  MoveL 2659 to (228.12, 35.85, 50.44) mm, rotated rx -180 ry 0 rz -180 deg; joints [-156.181, -75.797, -46.821, 39.316, 39.597, -32.253]
  MoveL 2660 to (228.12, 35.85, 50.44) mm, rotated rx -180 ry 0 rz -180 deg; joints [-156.181, -75.797, -46.821, 39.316, 39.597, -32.253]
  Call Extruder(588.66808)
  MoveL 2661 to (228.37, 35.9, 50.44) mm, rotated rx 180 ry 0 rz -180 deg; joints [-156.187, -75.828, -46.752, 39.337, 39.565, -32.285]
  MoveL 2662 to (228.37, 35.9, 50.44) mm, rotated rx 180 ry 0 rz -180 deg; joints [-156.187, -75.828, -46.752, 39.337, 39.565, -32.285]
  Call Extruder(588.80265)
  MoveL 2663 to (228.61, 35.95, 50.44) mm, rotated rx -180 ry 0 rz 180 deg; joints [-156.192, -75.86, -46.683, 39.359, 39.533, -32.317]
  MoveL 2664 to (228.61, 35.95, 50.44) mm, rotated rx -180 ry 0 rz 180 deg; joints [-156.192, -75.86, -46.683, 39.359, 39.533, -32.317]
  Call Extruder(588.88871)
  MoveL 2665 to (228.77, 35.98, 50.44) mm, rotated rx -180 ry 0 rz 180 deg; joints [-156.196, -75.88, -46.639, 39.373, 39.513, -32.338]
  MoveL 2666 to (228.77, 35.98, 50.44) mm, rotated rx -180 ry 0 rz 180 deg; joints [-156.196, -75.88, -46.639, 39.373, 39.513, -32.338]
  Call Extruder(589.00224)
  MoveL 2667 to (228.97, 36.02, 50.44) mm, rotated rx 180 ry 0 rz -180 deg; joints [-156.2, -75.906, -46.581, 39.391, 39.486, -32.365]
  MoveL 2668 to (228.97, 36.02, 50.44) mm, rotated rx 180 ry 0 rz -180 deg; joints [-156.2, -75.906, -46.581, 39.391, 39.486, -32.365]
  Call Extruder(589.11625)
  MoveL 2669 to (229.18, 36.06, 50.44) mm, rotated rx 180 ry 0 rz 180 deg; joints [-156.205, -75.932, -46.523, 39.41, 39.458, -32.392]
  MoveL 2670 to (229.18, 36.06, 50.44) mm, rotated rx 180 ry 0 rz 180 deg; joints [-156.205, -75.932, -46.523, 39.41, 39.458, -32.392]
  Call Extruder(589.23074)
  MoveL 2671 to (229.38, 36.1, 50.44) mm, rotated rx 180 ry 0 rz 180 deg; joints [-156.21, -75.958, -46.465, 39.428, 39.431, -32.419]
  MoveL 2672 to (229.38, 36.1, 50.44) mm, rotated rx 180 ry 0 rz 180 deg; joints [-156.21, -75.958, -46.465, 39.428, 39.431, -32.419]
  Call Extruder(589.35620)
  MoveL 2673 to (229.6, 36.16, 50.44) mm, rotated rx 180 ry 0 rz 180 deg; joints [-156.213, -75.988, -46.4, 39.451, 39.403, -32.451]
  MoveL 2674 to (229.6, 36.16, 50.44) mm, rotated rx 180 ry 0 rz 180 deg; joints [-156.213, -75.988, -46.4, 39.451, 39.403, -32.451]
  Call Extruder(589.48218)
  MoveL 2675 to (229.82, 36.23, 50.44) mm, rotated rx 180 ry 0 rz 180 deg; joints [-156.215, -76.017, -46.335, 39.475, 39.374, -32.483]
  MoveL 2676 to (229.82, 36.23, 50.44) mm, rotated rx 180 ry 0 rz 180 deg; joints [-156.215, -76.017, -46.335, 39.475, 39.374, -32.483]
  Call Extruder(589.60868)
  MoveL 2677 to (230.04, 36.29, 50.44) mm, rotated rx 180 ry 0 rz 180 deg; joints [-156.218, -76.046, -46.271, 39.498, 39.345, -32.516]
  MoveL 2678 to (230.04, 36.29, 50.44) mm, rotated rx 180 ry 0 rz 180 deg; joints [-156.218, -76.046, -46.271, 39.498, 39.345, -32.516]
  Call Extruder(589.73571)
  MoveL 2679 to (230.26, 36.36, 50.44) mm, rotated rx -180 ry 0 rz 180 deg; joints [-156.221, -76.076, -46.206, 39.522, 39.316, -32.549]
  MoveL 2680 to (230.26, 36.36, 50.44) mm, rotated rx -180 ry 0 rz 180 deg; joints [-156.221, -76.076, -46.206, 39.522, 39.316, -32.549]
  Call Extruder(589.86325)
  MoveL 2681 to (230.48, 36.42, 50.44) mm, rotated rx 180 ry 0 rz -180 deg; joints [-156.224, -76.105, -46.141, 39.546, 39.287, -32.581]
  MoveL 2682 to (230.48, 36.42, 50.44) mm, rotated rx 180 ry 0 rz -180 deg; joints [-156.224, -76.105, -46.141, 39.546, 39.287, -32.581]
  Call Extruder(589.99132)
  MoveL 2683 to (230.69, 36.49, 50.44) mm, rotated rx 180 ry 0 rz -180 deg; joints [-156.227, -76.135, -46.076, 39.57, 39.258, -32.614]
  MoveL 2684 to (230.69, 36.49, 50.44) mm, rotated rx 180 ry 0 rz -180 deg; joints [-156.227, -76.135, -46.076, 39.57, 39.258, -32.614]
  Call Extruder(590.10322)
  MoveL 2685 to (230.88, 36.55, 50.44) mm, rotated rx -180 ry 0 rz 180 deg; joints [-156.229, -76.161, -46.019, 39.591, 39.233, -32.643]
  MoveL 2686 to (230.88, 36.55, 50.44) mm, rotated rx -180 ry 0 rz 180 deg; joints [-156.229, -76.161, -46.019, 39.591, 39.233, -32.643]
  Call Extruder(590.21556)
  MoveL 2687 to (231.07, 36.61, 50.44) mm, rotated rx 180 ry 0 rz 180 deg; joints [-156.231, -76.186, -45.962, 39.613, 39.208, -32.672]
  MoveL 2688 to (231.07, 36.61, 50.44) mm, rotated rx 180 ry 0 rz 180 deg; joints [-156.231, -76.186, -45.962, 39.613, 39.208, -32.672]
  Call Extruder(590.32835)
  MoveL 2689 to (231.26, 36.67, 50.44) mm, rotated rx 180 ry 0 rz -180 deg; joints [-156.233, -76.212, -45.905, 39.634, 39.183, -32.702]
  MoveL 2690 to (231.26, 36.67, 50.44) mm, rotated rx 180 ry 0 rz -180 deg; joints [-156.233, -76.212, -45.905, 39.634, 39.183, -32.702]
  Call Extruder(590.44158)
  MoveL 2691 to (231.45, 36.73, 50.44) mm, rotated rx -180 ry 0 rz 180 deg; joints [-156.235, -76.238, -45.848, 39.656, 39.158, -32.731]
  MoveL 2692 to (231.45, 36.73, 50.44) mm, rotated rx -180 ry 0 rz 180 deg; joints [-156.235, -76.238, -45.848, 39.656, 39.158, -32.731]
  Call Extruder(590.55526)
  MoveL 2693 to (231.64, 36.79, 50.44) mm, rotated rx 180 ry 0 rz 180 deg; joints [-156.237, -76.264, -45.792, 39.678, 39.133, -32.76]
  MoveL 2694 to (231.64, 36.79, 50.44) mm, rotated rx 180 ry 0 rz 180 deg; joints [-156.237, -76.264, -45.792, 39.678, 39.133, -32.76]
  Call Extruder(590.73722)
  MoveL 2695 to (231.93, 36.91, 50.44) mm, rotated rx 180 ry 0 rz 180 deg; joints [-156.238, -76.306, -45.7, 39.716, 39.095, -32.81]
  MoveL 2696 to (231.93, 36.91, 50.44) mm, rotated rx 180 ry 0 rz 180 deg; joints [-156.238, -76.306, -45.7, 39.716, 39.095, -32.81]
  Call Extruder(590.91994)
  MoveL 2697 to (232.22, 37.03, 50.44) mm, rotated rx 180 ry 0 rz 180 deg; joints [-156.238, -76.347, -45.609, 39.754, 39.056, -32.86]
  MoveL 2698 to (232.22, 37.03, 50.44) mm, rotated rx 180 ry 0 rz 180 deg; joints [-156.238, -76.347, -45.609, 39.754, 39.056, -32.86]
  Call Extruder(591.09035)
  MoveL 2699 to (232.49, 37.15, 50.44) mm, rotated rx 180 ry 0 rz 180 deg; joints [-156.239, -76.386, -45.524, 39.79, 39.02, -32.906]
  MoveL 2700 to (232.49, 37.15, 50.44) mm, rotated rx 180 ry 0 rz 180 deg; joints [-156.239, -76.386, -45.524, 39.79, 39.02, -32.906]
  Call Extruder(591.24835)
  MoveL 2701 to (232.74, 37.26, 50.44) mm, rotated rx 180 ry 0 rz 180 deg; joints [-156.239, -76.422, -45.445, 39.824, 38.987, -32.95]
  MoveL 2702 to (232.74, 37.26, 50.44) mm, rotated rx 180 ry 0 rz 180 deg; joints [-156.239, -76.422, -45.445, 39.824, 38.987, -32.95]
  Call Extruder(591.40695)
  MoveL 2703 to (232.99, 37.36, 50.44) mm, rotated rx -180 ry 0 rz -180 deg; joints [-156.239, -76.458, -45.366, 39.858, 38.954, -32.993]
  MoveL 2704 to (232.99, 37.36, 50.44) mm, rotated rx -180 ry 0 rz -180 deg; joints [-156.239, -76.458, -45.366, 39.858, 38.954, -32.993]
  Call Extruder(591.61312)
  MoveL 2705 to (233.29, 37.54, 50.44) mm, rotated rx 180 ry 0 rz 180 deg; joints [-156.236, -76.504, -45.264, 39.906, 38.913, -33.054]
  MoveL 2706 to (233.29, 37.54, 50.44) mm, rotated rx 180 ry 0 rz 180 deg; joints [-156.236, -76.504, -45.264, 39.906, 38.913, -33.054]
  Call Extruder(591.82006)
  MoveL 2707 to (233.6, 37.71, 50.44) mm, rotated rx 180 ry 0 rz 180 deg; joints [-156.232, -76.55, -45.162, 39.956, 38.873, -33.114]
  MoveL 2708 to (233.6, 37.71, 50.44) mm, rotated rx 180 ry 0 rz 180 deg; joints [-156.232, -76.55, -45.162, 39.956, 38.873, -33.114]
  Call Extruder(592.02779)
  MoveL 2709 to (233.9, 37.89, 50.44) mm, rotated rx 180 ry 0 rz 180 deg; joints [-156.228, -76.597, -45.061, 40.005, 38.832, -33.175]
  MoveL 2710 to (233.9, 37.89, 50.44) mm, rotated rx 180 ry 0 rz 180 deg; joints [-156.228, -76.597, -45.061, 40.005, 38.832, -33.175]
  Call Extruder(592.23629)
  MoveL 2711 to (234.21, 38.06, 50.44) mm, rotated rx -180 ry 0 rz 180 deg; joints [-156.224, -76.643, -44.958, 40.054, 38.792, -33.236]
  MoveL 2712 to (234.21, 38.06, 50.44) mm, rotated rx -180 ry 0 rz 180 deg; joints [-156.224, -76.643, -44.958, 40.054, 38.792, -33.236]
  Call Extruder(592.41583)
  MoveL 2713 to (234.45, 38.24, 50.44) mm, rotated rx -180 ry 0 rz -180 deg; joints [-156.218, -76.683, -44.872, 40.1, 38.759, -33.291]
  MoveL 2714 to (234.45, 38.24, 50.44) mm, rotated rx -180 ry 0 rz -180 deg; joints [-156.218, -76.683, -44.872, 40.1, 38.759, -33.291]
  Call Extruder(592.74925)
  MoveL 2715 to (234.9, 38.57, 50.44) mm, rotated rx 180 ry 0 rz 180 deg; joints [-156.206, -76.756, -44.712, 40.186, 38.699, -33.393]
  MoveL 2716 to (234.9, 38.57, 50.44) mm, rotated rx 180 ry 0 rz 180 deg; joints [-156.206, -76.756, -44.712, 40.186, 38.699, -33.393]
  Call Extruder(593.08385)
  MoveL 2717 to (235.35, 38.9, 50.44) mm, rotated rx -180 ry 0 rz -180 deg; joints [-156.195, -76.829, -44.551, 40.272, 38.639, -33.495]
  Call Extruder(593.91180)
  MoveL 2718 to (236.39, 39.81, 50.44) mm, rotated rx -180 ry 0 rz 180 deg; joints [-156.154, -77.008, -44.161, 40.499, 38.501, -33.758]
  Call Extruder(594.73974)
  MoveL 2719 to (237.3, 40.85, 50.44) mm, rotated rx 180 ry 0 rz 180 deg; joints [-156.097, -77.178, -43.788, 40.741, 38.379, -34.029]
  Call Extruder(594.90704)
  MoveL 2720 to (237.47, 41.07, 50.44) mm, rotated rx 180 ry 0 rz 180 deg; joints [-156.083, -77.212, -43.716, 40.792, 38.357, -34.085]
  MoveL 2721 to (237.47, 41.07, 50.44) mm, rotated rx 180 ry 0 rz 180 deg; joints [-156.083, -77.212, -43.716, 40.792, 38.357, -34.085]
  Call Extruder(595.24045)
  MoveL 2722 to (237.8, 41.52, 50.44) mm, rotated rx -180 ry 0 rz 180 deg; joints [-156.055, -77.278, -43.571, 40.893, 38.313, -34.196]
  MoveL 2723 to (237.8, 41.52, 50.44) mm, rotated rx -180 ry 0 rz 180 deg; joints [-156.055, -77.278, -43.571, 40.893, 38.313, -34.196]
  Call Extruder(595.57268)
  MoveL 2724 to (238.12, 41.98, 50.44) mm, rotated rx 180 ry 0 rz -180 deg; joints [-156.028, -77.344, -43.426, 40.995, 38.269, -34.308]
  MoveL 2725 to (238.12, 41.98, 50.44) mm, rotated rx 180 ry 0 rz -180 deg; joints [-156.028, -77.344, -43.426, 40.995, 38.269, -34.308]
  Call Extruder(595.69039)
  MoveL 2726 to (238.22, 42.15, 50.44) mm, rotated rx -180 ry 0 rz 180 deg; joints [-156.016, -77.367, -43.378, 41.032, 38.256, -34.348]
  MoveL 2727 to (238.22, 42.15, 50.44) mm, rotated rx -180 ry 0 rz 180 deg; joints [-156.016, -77.367, -43.378, 41.032, 38.256, -34.348]
  Call Extruder(595.89811)
  MoveL 2728 to (238.4, 42.45, 50.44) mm, rotated rx 180 ry 0 rz 180 deg; joints [-155.996, -77.406, -43.292, 41.097, 38.232, -34.418]
  MoveL 2729 to (238.4, 42.45, 50.44) mm, rotated rx 180 ry 0 rz 180 deg; joints [-155.996, -77.406, -43.292, 41.097, 38.232, -34.418]
  Call Extruder(596.10507)
  MoveL 2730 to (238.57, 42.75, 50.44) mm, rotated rx 180 ry 0 rz -180 deg; joints [-155.976, -77.445, -43.207, 41.163, 38.209, -34.488]
  MoveL 2731 to (238.57, 42.75, 50.44) mm, rotated rx 180 ry 0 rz -180 deg; joints [-155.976, -77.445, -43.207, 41.163, 38.209, -34.488]
  Call Extruder(596.31124)
  MoveL 2732 to (238.75, 43.06, 50.44) mm, rotated rx 180 ry 0 rz 180 deg; joints [-155.956, -77.484, -43.121, 41.229, 38.186, -34.559]
  MoveL 2733 to (238.75, 43.06, 50.44) mm, rotated rx 180 ry 0 rz 180 deg; joints [-155.956, -77.484, -43.121, 41.229, 38.186, -34.559]
  Call Extruder(596.49292)
  MoveL 2734 to (238.89, 43.33, 50.44) mm, rotated rx -180 ry 0 rz -180 deg; joints [-155.937, -77.518, -43.048, 41.287, 38.167, -34.621]
  MoveL 2735 to (238.89, 43.33, 50.44) mm, rotated rx -180 ry 0 rz -180 deg; joints [-155.937, -77.518, -43.048, 41.287, 38.167, -34.621]
  Call Extruder(596.65093)
  MoveL 2736 to (239, 43.58, 50.44) mm, rotated rx -180 ry 0 rz -180 deg; joints [-155.919, -77.546, -42.988, 41.339, 38.153, -34.675]
  MoveL 2737 to (239, 43.58, 50.44) mm, rotated rx -180 ry 0 rz -180 deg; joints [-155.919, -77.546, -42.988, 41.339, 38.153, -34.675]
  Call Extruder(596.80833)
  MoveL 2738 to (239.11, 43.83, 50.44) mm, rotated rx 180 ry 0 rz -180 deg; joints [-155.901, -77.573, -42.927, 41.39, 38.138, -34.729]
  MoveL 2739 to (239.11, 43.83, 50.44) mm, rotated rx 180 ry 0 rz -180 deg; joints [-155.901, -77.573, -42.927, 41.39, 38.138, -34.729]
  Call Extruder(596.98254)
  MoveL 2740 to (239.22, 44.11, 50.44) mm, rotated rx 180 ry 0 rz 180 deg; joints [-155.88, -77.604, -42.861, 41.447, 38.123, -34.788]
  MoveL 2741 to (239.22, 44.11, 50.44) mm, rotated rx 180 ry 0 rz 180 deg; joints [-155.88, -77.604, -42.861, 41.447, 38.123, -34.788]
  Call Extruder(597.15607)
  MoveL 2742 to (239.33, 44.39, 50.44) mm, rotated rx 180 ry 0 rz 180 deg; joints [-155.86, -77.635, -42.794, 41.505, 38.108, -34.848]
  MoveL 2743 to (239.33, 44.39, 50.44) mm, rotated rx 180 ry 0 rz 180 deg; joints [-155.86, -77.635, -42.794, 41.505, 38.108, -34.848]
  Call Extruder(597.26356)
  MoveL 2744 to (239.41, 44.56, 50.44) mm, rotated rx 180 ry 0 rz -180 deg; joints [-155.847, -77.654, -42.753, 41.54, 38.098, -34.885]
  MoveL 2745 to (239.41, 44.56, 50.44) mm, rotated rx 180 ry 0 rz -180 deg; joints [-155.847, -77.654, -42.753, 41.54, 38.098, -34.885]
  Call Extruder(597.37703)
  MoveL 2746 to (239.47, 44.75, 50.44) mm, rotated rx 180 ry 0 rz -180 deg; joints [-155.833, -77.672, -42.713, 41.578, 38.09, -34.924]
  MoveL 2747 to (239.47, 44.75, 50.44) mm, rotated rx 180 ry 0 rz -180 deg; joints [-155.833, -77.672, -42.713, 41.578, 38.09, -34.924]
  Call Extruder(597.49005)
  MoveL 2748 to (239.53, 44.94, 50.44) mm, rotated rx 180 ry 0 rz 180 deg; joints [-155.819, -77.691, -42.672, 41.616, 38.082, -34.962]
  MoveL 2749 to (239.53, 44.94, 50.44) mm, rotated rx 180 ry 0 rz 180 deg; joints [-155.819, -77.691, -42.672, 41.616, 38.082, -34.962]
  Call Extruder(597.60263)
  MoveL 2750 to (239.59, 45.13, 50.44) mm, rotated rx 180 ry 0 rz -180 deg; joints [-155.804, -77.709, -42.632, 41.653, 38.074, -35.001]
  MoveL 2751 to (239.59, 45.13, 50.44) mm, rotated rx 180 ry 0 rz -180 deg; joints [-155.804, -77.709, -42.632, 41.653, 38.074, -35.001]
  Call Extruder(597.71477)
  MoveL 2752 to (239.65, 45.32, 50.44) mm, rotated rx 180 ry 0 rz 180 deg; joints [-155.79, -77.728, -42.591, 41.691, 38.066, -35.04]
  MoveL 2753 to (239.65, 45.32, 50.44) mm, rotated rx 180 ry 0 rz 180 deg; joints [-155.79, -77.728, -42.591, 41.691, 38.066, -35.04]
  Call Extruder(597.82645)
  MoveL 2754 to (239.71, 45.5, 50.44) mm, rotated rx -180 ry 0 rz 180 deg; joints [-155.776, -77.747, -42.55, 41.728, 38.058, -35.078]
  MoveL 2755 to (239.71, 45.5, 50.44) mm, rotated rx -180 ry 0 rz 180 deg; joints [-155.776, -77.747, -42.55, 41.728, 38.058, -35.078]
  Call Extruder(597.95753)
  MoveL 2756 to (239.78, 45.73, 50.44) mm, rotated rx 180 ry 0 rz 180 deg; joints [-155.758, -77.768, -42.504, 41.773, 38.049, -35.124]
  MoveL 2757 to (239.78, 45.73, 50.44) mm, rotated rx 180 ry 0 rz 180 deg; joints [-155.758, -77.768, -42.504, 41.773, 38.049, -35.124]
  Call Extruder(598.08804)
  MoveL 2758 to (239.85, 45.95, 50.44) mm, rotated rx 180 ry 0 rz 180 deg; joints [-155.741, -77.79, -42.457, 41.817, 38.04, -35.169]
  MoveL 2759 to (239.85, 45.95, 50.44) mm, rotated rx 180 ry 0 rz 180 deg; joints [-155.741, -77.79, -42.457, 41.817, 38.04, -35.169]
  Call Extruder(598.21798)
  MoveL 2760 to (239.92, 46.18, 50.44) mm, rotated rx -180 ry 0 rz 180 deg; joints [-155.724, -77.812, -42.41, 41.862, 38.031, -35.214]
  MoveL 2761 to (239.92, 46.18, 50.44) mm, rotated rx -180 ry 0 rz 180 deg; joints [-155.724, -77.812, -42.41, 41.862, 38.031, -35.214]
  Call Extruder(598.34736)
  MoveL 2762 to (239.98, 46.4, 50.44) mm, rotated rx 180 ry 0 rz 180 deg; joints [-155.707, -77.833, -42.363, 41.906, 38.022, -35.26]
  MoveL 2763 to (239.98, 46.4, 50.44) mm, rotated rx 180 ry 0 rz 180 deg; joints [-155.707, -77.833, -42.363, 41.906, 38.022, -35.26]
  Call Extruder(598.46931)
  MoveL 2764 to (240.04, 46.61, 50.44) mm, rotated rx 180 ry 0 rz -180 deg; joints [-155.69, -77.853, -42.32, 41.948, 38.014, -35.302]
  MoveL 2765 to (240.04, 46.61, 50.44) mm, rotated rx 180 ry 0 rz -180 deg; joints [-155.69, -77.853, -42.32, 41.948, 38.014, -35.302]
  Call Extruder(598.58414)
  MoveL 2766 to (240.08, 46.82, 50.44) mm, rotated rx 180 ry 0 rz -180 deg; joints [-155.674, -77.87, -42.282, 41.987, 38.009, -35.342]
  MoveL 2767 to (240.08, 46.82, 50.44) mm, rotated rx 180 ry 0 rz -180 deg; joints [-155.674, -77.87, -42.282, 41.987, 38.009, -35.342]
  Call Extruder(598.69851)
  MoveL 2768 to (240.13, 47.02, 50.44) mm, rotated rx -180 ry 0 rz 180 deg; joints [-155.657, -77.888, -42.244, 42.027, 38.003, -35.381]
  MoveL 2769 to (240.13, 47.02, 50.44) mm, rotated rx -180 ry 0 rz 180 deg; joints [-155.657, -77.888, -42.244, 42.027, 38.003, -35.381]
  Call Extruder(598.81243)
  MoveL 2770 to (240.17, 47.23, 50.44) mm, rotated rx 180 ry 0 rz 180 deg; joints [-155.641, -77.906, -42.205, 42.066, 37.997, -35.421]
  MoveL 2771 to (240.17, 47.23, 50.44) mm, rotated rx 180 ry 0 rz 180 deg; joints [-155.641, -77.906, -42.205, 42.066, 37.997, -35.421]
  Call Extruder(598.92591)
  MoveL 2772 to (240.22, 47.43, 50.44) mm, rotated rx -180 ry 0 rz 180 deg; joints [-155.624, -77.923, -42.167, 42.105, 37.991, -35.46]
  MoveL 2773 to (240.22, 47.43, 50.44) mm, rotated rx -180 ry 0 rz 180 deg; joints [-155.624, -77.923, -42.167, 42.105, 37.991, -35.46]
  Call Extruder(599.06319)
  MoveL 2774 to (240.27, 47.68, 50.44) mm, rotated rx 180 ry 0 rz 180 deg; joints [-155.604, -77.944, -42.122, 42.153, 37.985, -35.508]
  MoveL 2775 to (240.27, 47.68, 50.44) mm, rotated rx 180 ry 0 rz 180 deg; joints [-155.604, -77.944, -42.122, 42.153, 37.985, -35.508]
  Call Extruder(599.19986)
  MoveL 2776 to (240.32, 47.93, 50.44) mm, rotated rx 180 ry 0 rz -180 deg; joints [-155.584, -77.965, -42.076, 42.201, 37.978, -35.556]
  MoveL 2777 to (240.32, 47.93, 50.44) mm, rotated rx 180 ry 0 rz -180 deg; joints [-155.584, -77.965, -42.076, 42.201, 37.978, -35.556]
  Call Extruder(599.33592)
  MoveL 2778 to (240.37, 48.18, 50.44) mm, rotated rx 180 ry 0 rz 180 deg; joints [-155.564, -77.986, -42.031, 42.249, 37.972, -35.603]
  MoveL 2779 to (240.37, 48.18, 50.44) mm, rotated rx 180 ry 0 rz 180 deg; joints [-155.564, -77.986, -42.031, 42.249, 37.972, -35.603]
  Call Extruder(599.47137)
  MoveL 2780 to (240.42, 48.43, 50.44) mm, rotated rx 180 ry 0 rz 180 deg; joints [-155.544, -78.007, -41.985, 42.296, 37.965, -35.651]
  MoveL 2781 to (240.42, 48.43, 50.44) mm, rotated rx 180 ry 0 rz 180 deg; joints [-155.544, -78.007, -41.985, 42.296, 37.965, -35.651]
  Call Extruder(599.60622)
  MoveL 2782 to (240.47, 48.68, 50.44) mm, rotated rx 180 ry 0 rz 180 deg; joints [-155.524, -78.028, -41.939, 42.344, 37.959, -35.699]
  MoveL 2783 to (240.47, 48.68, 50.44) mm, rotated rx 180 ry 0 rz 180 deg; joints [-155.524, -78.028, -41.939, 42.344, 37.959, -35.699]
  Call Extruder(599.74045)
  MoveL 2784 to (240.52, 48.92, 50.44) mm, rotated rx 180 ry 0 rz 180 deg; joints [-155.504, -78.05, -41.893, 42.392, 37.952, -35.747]
  MoveL 2785 to (240.52, 48.92, 50.44) mm, rotated rx 180 ry 0 rz 180 deg; joints [-155.504, -78.05, -41.893, 42.392, 37.952, -35.747]
  Call Extruder(599.87407)
  MoveL 2786 to (240.56, 49.17, 50.44) mm, rotated rx -180 ry 0 rz 180 deg; joints [-155.484, -78.071, -41.848, 42.44, 37.946, -35.795]
  MoveL 2787 to (240.56, 49.17, 50.44) mm, rotated rx -180 ry 0 rz 180 deg; joints [-155.484, -78.071, -41.848, 42.44, 37.946, -35.795]
  Call Extruder(600.03618)
  MoveL 2788 to (240.61, 49.48, 50.44) mm, rotated rx -180 ry 0 rz 180 deg; joints [-155.459, -78.095, -41.795, 42.497, 37.939, -35.852]
  MoveL 2789 to (240.61, 49.48, 50.44) mm, rotated rx -180 ry 0 rz 180 deg; joints [-155.459, -78.095, -41.795, 42.497, 37.939, -35.852]
  Call Extruder(600.19756)
  MoveL 2790 to (240.66, 49.79, 50.44) mm, rotated rx 180 ry 0 rz 180 deg; joints [-155.433, -78.12, -41.742, 42.555, 37.933, -35.91]
  MoveL 2791 to (240.66, 49.79, 50.44) mm, rotated rx 180 ry 0 rz 180 deg; joints [-155.433, -78.12, -41.742, 42.555, 37.933, -35.91]
  Call Extruder(600.35821)
  MoveL 2792 to (240.71, 50.09, 50.44) mm, rotated rx -180 ry 0 rz 180 deg; joints [-155.408, -78.144, -41.689, 42.613, 37.927, -35.967]
  MoveL 2793 to (240.71, 50.09, 50.44) mm, rotated rx -180 ry 0 rz 180 deg; joints [-155.408, -78.144, -41.689, 42.613, 37.927, -35.967]
  Call Extruder(600.51814)
  MoveL 2794 to (240.76, 50.4, 50.44) mm, rotated rx 180 ry 0 rz 180 deg; joints [-155.383, -78.169, -41.636, 42.671, 37.921, -36.025]
  MoveL 2795 to (240.76, 50.4, 50.44) mm, rotated rx 180 ry 0 rz 180 deg; joints [-155.383, -78.169, -41.636, 42.671, 37.921, -36.025]
  Call Extruder(600.67734)
  MoveL 2796 to (240.81, 50.7, 50.44) mm, rotated rx -180 ry 0 rz 180 deg; joints [-155.358, -78.193, -41.583, 42.729, 37.914, -36.082]
  MoveL 2797 to (240.81, 50.7, 50.44) mm, rotated rx -180 ry 0 rz 180 deg; joints [-155.358, -78.193, -41.583, 42.729, 37.914, -36.082]
  Call Extruder(600.83580)
  MoveL 2798 to (240.86, 51.01, 50.44) mm, rotated rx 180 ry 0 rz -180 deg; joints [-155.333, -78.218, -41.529, 42.787, 37.908, -36.14]
  MoveL 2799 to (240.86, 51.01, 50.44) mm, rotated rx 180 ry 0 rz -180 deg; joints [-155.333, -78.218, -41.529, 42.787, 37.908, -36.14]
  Call Extruder(601.03468)
  MoveL 2800 to (240.9, 51.4, 50.44) mm, rotated rx -180 ry 0 rz -180 deg; joints [-155.301, -78.247, -41.466, 42.859, 37.902, -36.211]
  MoveL 2801 to (240.9, 51.4, 50.44) mm, rotated rx -180 ry 0 rz -180 deg; joints [-155.301, -78.247, -41.466, 42.859, 37.902, -36.211]
  Call Extruder(601.23269)
  MoveL 2802 to (240.95, 51.78, 50.44) mm, rotated rx 180 ry 0 rz 180 deg; joints [-155.268, -78.276, -41.403, 42.931, 37.896, -36.282]
  MoveL 2803 to (240.95, 51.78, 50.44) mm, rotated rx 180 ry 0 rz 180 deg; joints [-155.268, -78.276, -41.403, 42.931, 37.896, -36.282]
  Call Extruder(601.42983)
  MoveL 2804 to (240.99, 52.17, 50.44) mm, rotated rx 180 ry 0 rz 180 deg; joints [-155.236, -78.306, -41.339, 43.003, 37.891, -36.354]
  MoveL 2805 to (240.99, 52.17, 50.44) mm, rotated rx 180 ry 0 rz 180 deg; joints [-155.236, -78.306, -41.339, 43.003, 37.891, -36.354]
  Call Extruder(601.62610)
  MoveL 2806 to (241.04, 52.56, 50.44) mm, rotated rx 180 ry 0 rz 180 deg; joints [-155.204, -78.335, -41.276, 43.076, 37.885, -36.425]
  MoveL 2807 to (241.04, 52.56, 50.44) mm, rotated rx 180 ry 0 rz 180 deg; joints [-155.204, -78.335, -41.276, 43.076, 37.885, -36.425]
  Call Extruder(601.87181)
  MoveL 2808 to (241.09, 53.05, 50.44) mm, rotated rx 180 ry 0 rz 180 deg; joints [-155.163, -78.371, -41.199, 43.166, 37.879, -36.514]
  MoveL 2809 to (241.09, 53.05, 50.44) mm, rotated rx 180 ry 0 rz 180 deg; joints [-155.163, -78.371, -41.199, 43.166, 37.879, -36.514]
  Call Extruder(602.16658)
  MoveL 2810 to (241.13, 53.64, 50.44) mm, rotated rx 180 ry 0 rz 180 deg; joints [-155.113, -78.413, -41.108, 43.274, 37.873, -36.62]
  MoveL 2811 to (241.13, 53.64, 50.44) mm, rotated rx 180 ry 0 rz 180 deg; joints [-155.113, -78.413, -41.108, 43.274, 37.873, -36.62]
  Call Extruder(602.46002)
  MoveL 2812 to (241.18, 54.23, 50.44) mm, rotated rx 180 ry 0 rz 180 deg; joints [-155.063, -78.455, -41.017, 43.383, 37.868, -36.726]
  MoveL 2813 to (241.18, 54.23, 50.44) mm, rotated rx 180 ry 0 rz 180 deg; joints [-155.063, -78.455, -41.017, 43.383, 37.868, -36.726]
  Call Extruder(602.89337)
  MoveL 2814 to (241.22, 55.1, 50.44) mm, rotated rx 180 ry 0 rz -180 deg; joints [-154.988, -78.514, -40.888, 43.542, 37.862, -36.881]
  MoveL 2815 to (241.22, 55.1, 50.44) mm, rotated rx 180 ry 0 rz -180 deg; joints [-154.988, -78.514, -40.888, 43.542, 37.862, -36.881]
  Call Extruder(603.46554)
  MoveL 2816 to (241.27, 56.27, 50.44) mm, rotated rx -180 ry 0 rz -180 deg; joints [-154.887, -78.592, -40.72, 43.752, 37.857, -37.085]
  MoveL 2817 to (241.27, 56.27, 50.44) mm, rotated rx -180 ry 0 rz -180 deg; joints [-154.887, -78.592, -40.72, 43.752, 37.857, -37.085]
  Call Extruder(603.89324)
  MoveL 2818 to (241.29, 57.14, 50.44) mm, rotated rx 180 ry 0 rz 180 deg; joints [-154.812, -78.649, -40.599, 43.909, 37.856, -37.236]
  Call Extruder(645.88687)
  MoveL 2819 to (241.29, 142.86, 50.44) mm, rotated rx -180 ry 0 rz 180 deg; joints [-147.778, -85.814, -25.526, 59.999, 38.002, -53.77]
  MoveL 2820 to (241.29, 142.86, 50.44) mm, rotated rx -180 ry 0 rz 180 deg; joints [-147.778, -85.814, -25.526, 59.999, 38.002, -53.77]
  Call Extruder(646.60231)
  MoveL 2821 to (241.25, 144.32, 50.44) mm, rotated rx -180 ry 0 rz -180 deg; joints [-147.665, -85.972, -25.201, 60.293, 38.01, -54.09]
  MoveL 2822 to (241.25, 144.32, 50.44) mm, rotated rx -180 ry 0 rz -180 deg; joints [-147.665, -85.972, -25.201, 60.293, 38.01, -54.09]
  Call Extruder(647.17705)
  MoveL 2823 to (241.2, 145.48, 50.44) mm, rotated rx 180 ry 0 rz -180 deg; joints [-147.574, -86.097, -24.944, 60.526, 38.019, -54.344]
  MoveL 2824 to (241.2, 145.48, 50.44) mm, rotated rx 180 ry 0 rz -180 deg; joints [-147.574, -86.097, -24.944, 60.526, 38.019, -54.344]
  Call Extruder(647.47049)
  MoveL 2825 to (241.16, 146.07, 50.44) mm, rotated rx -180 ry 0 rz 180 deg; joints [-147.527, -86.156, -24.822, 60.64, 38.026, -54.468]
  MoveL 2826 to (241.16, 146.07, 50.44) mm, rotated rx -180 ry 0 rz 180 deg; joints [-147.527, -86.156, -24.822, 60.64, 38.026, -54.468]
  Call Extruder(647.76527)
  MoveL 2827 to (241.11, 146.66, 50.44) mm, rotated rx -180 ry 0 rz -180 deg; joints [-147.48, -86.216, -24.699, 60.755, 38.034, -54.592]
  MoveL 2828 to (241.11, 146.66, 50.44) mm, rotated rx -180 ry 0 rz -180 deg; joints [-147.48, -86.216, -24.699, 60.755, 38.034, -54.592]
  Call Extruder(648.06138)
  MoveL 2829 to (241.06, 147.25, 50.44) mm, rotated rx -180 ry 0 rz 180 deg; joints [-147.433, -86.276, -24.575, 60.87, 38.041, -54.717]
  MoveL 2830 to (241.06, 147.25, 50.44) mm, rotated rx -180 ry 0 rz 180 deg; joints [-147.433, -86.276, -24.575, 60.87, 38.041, -54.717]
  Call Extruder(648.25765)
  MoveL 2831 to (241.02, 147.63, 50.44) mm, rotated rx 180 ry 0 rz 180 deg; joints [-147.401, -86.314, -24.499, 60.943, 38.048, -54.795]
  MoveL 2832 to (241.02, 147.63, 50.44) mm, rotated rx 180 ry 0 rz 180 deg; joints [-147.401, -86.314, -24.499, 60.943, 38.048, -54.795]
  Call Extruder(648.45479)
  MoveL 2833 to (240.97, 148.02, 50.44) mm, rotated rx 180 ry 0 rz -180 deg; joints [-147.37, -86.351, -24.423, 61.016, 38.055, -54.874]
  MoveL 2834 to (240.97, 148.02, 50.44) mm, rotated rx 180 ry 0 rz -180 deg; joints [-147.37, -86.351, -24.423, 61.016, 38.055, -54.874]
  Call Extruder(648.65280)
  MoveL 2835 to (240.92, 148.41, 50.44) mm, rotated rx 180 ry 0 rz -180 deg; joints [-147.338, -86.388, -24.347, 61.089, 38.062, -54.952]
  MoveL 2836 to (240.92, 148.41, 50.44) mm, rotated rx 180 ry 0 rz -180 deg; joints [-147.338, -86.388, -24.347, 61.089, 38.062, -54.952]
  Call Extruder(648.85167)
  MoveL 2837 to (240.88, 148.8, 50.44) mm, rotated rx -180 ry 0 rz -180 deg; joints [-147.306, -86.425, -24.27, 61.162, 38.069, -55.031]
  MoveL 2838 to (240.88, 148.8, 50.44) mm, rotated rx -180 ry 0 rz -180 deg; joints [-147.306, -86.425, -24.27, 61.162, 38.069, -55.031]
  Call Extruder(649.03075)
  MoveL 2839 to (240.83, 149.14, 50.44) mm, rotated rx 180 ry 0 rz 180 deg; joints [-147.278, -86.458, -24.204, 61.227, 38.076, -55.1]
  MoveL 2840 to (240.83, 149.14, 50.44) mm, rotated rx 180 ry 0 rz 180 deg; joints [-147.278, -86.458, -24.204, 61.227, 38.076, -55.1]
  Call Extruder(649.18995)
  MoveL 2841 to (240.78, 149.45, 50.44) mm, rotated rx 180 ry 0 rz 180 deg; joints [-147.252, -86.485, -24.148, 61.283, 38.083, -55.16]
  MoveL 2842 to (240.78, 149.45, 50.44) mm, rotated rx 180 ry 0 rz 180 deg; joints [-147.252, -86.485, -24.148, 61.283, 38.083, -55.16]
  Call Extruder(649.34987)
  MoveL 2843 to (240.74, 149.76, 50.44) mm, rotated rx 180 ry 0 rz -180 deg; joints [-147.227, -86.512, -24.091, 61.339, 38.09, -55.22]
  MoveL 2844 to (240.74, 149.76, 50.44) mm, rotated rx 180 ry 0 rz -180 deg; joints [-147.227, -86.512, -24.091, 61.339, 38.09, -55.22]
  Call Extruder(649.51052)
  MoveL 2845 to (240.69, 150.06, 50.44) mm, rotated rx -180 ry 0 rz -180 deg; joints [-147.201, -86.54, -24.035, 61.394, 38.097, -55.279]
  MoveL 2846 to (240.69, 150.06, 50.44) mm, rotated rx -180 ry 0 rz -180 deg; joints [-147.201, -86.54, -24.035, 61.394, 38.097, -55.279]
  Call Extruder(649.67190)
  MoveL 2847 to (240.64, 150.37, 50.44) mm, rotated rx 180 ry 0 rz 180 deg; joints [-147.176, -86.568, -23.978, 61.45, 38.105, -55.339]
  MoveL 2848 to (240.64, 150.37, 50.44) mm, rotated rx 180 ry 0 rz 180 deg; joints [-147.176, -86.568, -23.978, 61.45, 38.105, -55.339]
  Call Extruder(649.83401)
  MoveL 2849 to (240.59, 150.67, 50.44) mm, rotated rx 180 ry 0 rz 180 deg; joints [-147.15, -86.595, -23.922, 61.506, 38.112, -55.398]
  MoveL 2850 to (240.59, 150.67, 50.44) mm, rotated rx 180 ry 0 rz 180 deg; joints [-147.15, -86.595, -23.922, 61.506, 38.112, -55.398]
  Call Extruder(649.98221)
  MoveL 2851 to (240.54, 150.95, 50.44) mm, rotated rx 180 ry 0 rz 180 deg; joints [-147.127, -86.619, -23.872, 61.556, 38.119, -55.451]
  MoveL 2852 to (240.54, 150.95, 50.44) mm, rotated rx 180 ry 0 rz 180 deg; joints [-147.127, -86.619, -23.872, 61.556, 38.119, -55.451]
  Call Extruder(650.11644)
  MoveL 2853 to (240.49, 151.2, 50.44) mm, rotated rx 180 ry 0 rz 180 deg; joints [-147.106, -86.64, -23.83, 61.6, 38.126, -55.498]
  MoveL 2854 to (240.49, 151.2, 50.44) mm, rotated rx 180 ry 0 rz 180 deg; joints [-147.106, -86.64, -23.83, 61.6, 38.126, -55.498]
  Call Extruder(650.25129)
  MoveL 2855 to (240.44, 151.45, 50.44) mm, rotated rx -180 ry 0 rz -180 deg; joints [-147.085, -86.661, -23.787, 61.644, 38.133, -55.544]
  MoveL 2856 to (240.44, 151.45, 50.44) mm, rotated rx -180 ry 0 rz -180 deg; joints [-147.085, -86.661, -23.787, 61.644, 38.133, -55.544]
  Call Extruder(650.38674)
  MoveL 2857 to (240.39, 151.7, 50.44) mm, rotated rx 180 ry 0 rz 180 deg; joints [-147.064, -86.682, -23.744, 61.688, 38.14, -55.591]
  MoveL 2858 to (240.39, 151.7, 50.44) mm, rotated rx 180 ry 0 rz 180 deg; joints [-147.064, -86.682, -23.744, 61.688, 38.14, -55.591]
  Call Extruder(650.52280)
  MoveL 2859 to (240.34, 151.95, 50.44) mm, rotated rx 180 ry 0 rz 180 deg; joints [-147.042, -86.703, -23.701, 61.732, 38.147, -55.637]
  MoveL 2860 to (240.34, 151.95, 50.44) mm, rotated rx 180 ry 0 rz 180 deg; joints [-147.042, -86.703, -23.701, 61.732, 38.147, -55.637]
  Call Extruder(650.65947)
  MoveL 2861 to (240.29, 152.2, 50.44) mm, rotated rx -180 ry 0 rz 180 deg; joints [-147.021, -86.724, -23.658, 61.776, 38.154, -55.684]
  MoveL 2862 to (240.29, 152.2, 50.44) mm, rotated rx -180 ry 0 rz 180 deg; joints [-147.021, -86.724, -23.658, 61.776, 38.154, -55.684]
  Call Extruder(650.79675)
  MoveL 2863 to (240.24, 152.44, 50.44) mm, rotated rx 180 ry 0 rz -180 deg; joints [-147, -86.745, -23.616, 61.82, 38.162, -55.73]
  MoveL 2864 to (240.24, 152.44, 50.44) mm, rotated rx 180 ry 0 rz -180 deg; joints [-147, -86.745, -23.616, 61.82, 38.162, -55.73]
  Call Extruder(650.92242)
  MoveL 2865 to (240.2, 152.67, 50.44) mm, rotated rx 180 ry 0 rz 180 deg; joints [-146.981, -86.764, -23.577, 61.859, 38.168, -55.772]
  MoveL 2866 to (240.2, 152.67, 50.44) mm, rotated rx 180 ry 0 rz 180 deg; joints [-146.981, -86.764, -23.577, 61.859, 38.168, -55.772]
  Call Extruder(651.03634)
  MoveL 2867 to (240.15, 152.88, 50.44) mm, rotated rx 180 ry 0 rz 180 deg; joints [-146.963, -86.78, -23.543, 61.895, 38.175, -55.809]
  MoveL 2868 to (240.15, 152.88, 50.44) mm, rotated rx 180 ry 0 rz 180 deg; joints [-146.963, -86.78, -23.543, 61.895, 38.175, -55.809]
  Call Extruder(651.15072)
  MoveL 2869 to (240.11, 153.08, 50.44) mm, rotated rx -180 ry 0 rz -180 deg; joints [-146.945, -86.797, -23.509, 61.93, 38.181, -55.847]
  MoveL 2870 to (240.11, 153.08, 50.44) mm, rotated rx -180 ry 0 rz -180 deg; joints [-146.945, -86.797, -23.509, 61.93, 38.181, -55.847]
  Call Extruder(651.26555)
  MoveL 2871 to (240.06, 153.28, 50.44) mm, rotated rx 180 ry 0 rz 180 deg; joints [-146.928, -86.813, -23.476, 61.965, 38.187, -55.884]
  MoveL 2872 to (240.06, 153.28, 50.44) mm, rotated rx 180 ry 0 rz 180 deg; joints [-146.928, -86.813, -23.476, 61.965, 38.187, -55.884]
  Call Extruder(651.38083)
  MoveL 2873 to (240.02, 153.49, 50.44) mm, rotated rx 180 ry 0 rz 180 deg; joints [-146.91, -86.83, -23.442, 62.001, 38.194, -55.921]
  MoveL 2874 to (240.02, 153.49, 50.44) mm, rotated rx 180 ry 0 rz 180 deg; joints [-146.91, -86.83, -23.442, 62.001, 38.194, -55.921]
  Call Extruder(651.51021)
  MoveL 2875 to (239.95, 153.71, 50.44) mm, rotated rx 180 ry 0 rz 180 deg; joints [-146.89, -86.845, -23.411, 62.036, 38.203, -55.957]
  MoveL 2876 to (239.95, 153.71, 50.44) mm, rotated rx 180 ry 0 rz 180 deg; joints [-146.89, -86.845, -23.411, 62.036, 38.203, -55.957]
  Call Extruder(651.64015)
  MoveL 2877 to (239.88, 153.94, 50.44) mm, rotated rx 180 ry 0 rz 180 deg; joints [-146.87, -86.859, -23.381, 62.072, 38.213, -55.994]
  MoveL 2878 to (239.88, 153.94, 50.44) mm, rotated rx 180 ry 0 rz 180 deg; joints [-146.87, -86.859, -23.381, 62.072, 38.213, -55.994]
  Call Extruder(651.77066)
  MoveL 2879 to (239.81, 154.16, 50.44) mm, rotated rx 180 ry 0 rz -180 deg; joints [-146.85, -86.874, -23.351, 62.107, 38.222, -56.03]
  MoveL 2880 to (239.81, 154.16, 50.44) mm, rotated rx 180 ry 0 rz -180 deg; joints [-146.85, -86.874, -23.351, 62.107, 38.222, -56.03]
  Call Extruder(651.90174)
  MoveL 2881 to (239.75, 154.38, 50.44) mm, rotated rx 180 ry 0 rz 180 deg; joints [-146.83, -86.889, -23.321, 62.143, 38.232, -56.066]
  MoveL 2882 to (239.75, 154.38, 50.44) mm, rotated rx 180 ry 0 rz 180 deg; joints [-146.83, -86.889, -23.321, 62.143, 38.232, -56.066]
  Call Extruder(652.02338)
  MoveL 2883 to (239.68, 154.59, 50.44) mm, rotated rx 180 ry 0 rz 180 deg; joints [-146.811, -86.902, -23.294, 62.175, 38.241, -56.099]
  MoveL 2884 to (239.68, 154.59, 50.44) mm, rotated rx 180 ry 0 rz 180 deg; joints [-146.811, -86.902, -23.294, 62.175, 38.241, -56.099]
  Call Extruder(652.13550)
  MoveL 2885 to (239.62, 154.78, 50.44) mm, rotated rx -180 ry 0 rz -180 deg; joints [-146.794, -86.914, -23.27, 62.204, 38.249, -56.129]
  MoveL 2886 to (239.62, 154.78, 50.44) mm, rotated rx -180 ry 0 rz -180 deg; joints [-146.794, -86.914, -23.27, 62.204, 38.249, -56.129]
  Call Extruder(652.24807)
  MoveL 2887 to (239.56, 154.97, 50.44) mm, rotated rx -180 ry 0 rz 180 deg; joints [-146.777, -86.926, -23.246, 62.234, 38.258, -56.159]
  MoveL 2888 to (239.56, 154.97, 50.44) mm, rotated rx -180 ry 0 rz 180 deg; joints [-146.777, -86.926, -23.246, 62.234, 38.258, -56.159]
  Call Extruder(652.36108)
  MoveL 2889 to (239.5, 155.15, 50.44) mm, rotated rx -180 ry 0 rz 180 deg; joints [-146.76, -86.937, -23.222, 62.263, 38.266, -56.188]
  MoveL 2890 to (239.5, 155.15, 50.44) mm, rotated rx -180 ry 0 rz 180 deg; joints [-146.76, -86.937, -23.222, 62.263, 38.266, -56.188]
  Call Extruder(652.47454)
  MoveL 2891 to (239.44, 155.34, 50.44) mm, rotated rx 180 ry 0 rz -180 deg; joints [-146.742, -86.949, -23.198, 62.292, 38.275, -56.218]
  MoveL 2892 to (239.44, 155.34, 50.44) mm, rotated rx 180 ry 0 rz -180 deg; joints [-146.742, -86.949, -23.198, 62.292, 38.275, -56.218]
  Call Extruder(652.62218)
  MoveL 2893 to (239.35, 155.58, 50.44) mm, rotated rx -180 ry 0 rz -180 deg; joints [-146.72, -86.962, -23.172, 62.327, 38.287, -56.253]
  MoveL 2894 to (239.35, 155.58, 50.44) mm, rotated rx -180 ry 0 rz -180 deg; joints [-146.72, -86.962, -23.172, 62.327, 38.287, -56.253]
  Call Extruder(652.80452)
  MoveL 2895 to (239.23, 155.87, 50.44) mm, rotated rx -180 ry 0 rz 180 deg; joints [-146.692, -86.975, -23.145, 62.368, 38.304, -56.292]
  MoveL 2896 to (239.23, 155.87, 50.44) mm, rotated rx -180 ry 0 rz 180 deg; joints [-146.692, -86.975, -23.145, 62.368, 38.304, -56.292]
  Call Extruder(652.98761)
  MoveL 2897 to (239.11, 156.17, 50.44) mm, rotated rx 180 ry 0 rz 180 deg; joints [-146.664, -86.989, -23.117, 62.408, 38.321, -56.332]
  MoveL 2898 to (239.11, 156.17, 50.44) mm, rotated rx 180 ry 0 rz 180 deg; joints [-146.664, -86.989, -23.117, 62.408, 38.321, -56.332]
  Call Extruder(653.14533)
  MoveL 2899 to (239, 156.42, 50.44) mm, rotated rx 180 ry 0 rz -180 deg; joints [-146.64, -87, -23.095, 62.442, 38.335, -56.365]
  MoveL 2900 to (239, 156.42, 50.44) mm, rotated rx 180 ry 0 rz -180 deg; joints [-146.64, -87, -23.095, 62.442, 38.335, -56.365]
  Call Extruder(653.30365)
  MoveL 2901 to (238.89, 156.66, 50.44) mm, rotated rx -180 ry 0 rz 180 deg; joints [-146.617, -87.01, -23.073, 62.476, 38.35, -56.398]
  MoveL 2902 to (238.89, 156.66, 50.44) mm, rotated rx -180 ry 0 rz 180 deg; joints [-146.617, -87.01, -23.073, 62.476, 38.35, -56.398]
  Call Extruder(653.48569)
  MoveL 2903 to (238.75, 156.94, 50.44) mm, rotated rx -180 ry 0 rz 180 deg; joints [-146.589, -87.018, -23.057, 62.51, 38.369, -56.429]
  MoveL 2904 to (238.75, 156.94, 50.44) mm, rotated rx -180 ry 0 rz 180 deg; joints [-146.589, -87.018, -23.057, 62.51, 38.369, -56.429]
  Call Extruder(653.69224)
  MoveL 2905 to (238.57, 157.25, 50.44) mm, rotated rx 180 ry 0 rz 180 deg; joints [-146.557, -87.023, -23.047, 62.544, 38.393, -56.458]
  MoveL 2906 to (238.57, 157.25, 50.44) mm, rotated rx 180 ry 0 rz 180 deg; joints [-146.557, -87.023, -23.047, 62.544, 38.393, -56.458]
  Call Extruder(653.89957)
  MoveL 2907 to (238.4, 157.55, 50.44) mm, rotated rx 180 ry 0 rz 180 deg; joints [-146.526, -87.028, -23.037, 62.577, 38.417, -56.487]
  MoveL 2908 to (238.4, 157.55, 50.44) mm, rotated rx 180 ry 0 rz 180 deg; joints [-146.526, -87.028, -23.037, 62.577, 38.417, -56.487]
  Call Extruder(654.10768)
  MoveL 2909 to (238.22, 157.85, 50.44) mm, rotated rx -180 ry 0 rz 180 deg; joints [-146.495, -87.033, -23.027, 62.611, 38.441, -56.516]
  MoveL 2910 to (238.22, 157.85, 50.44) mm, rotated rx -180 ry 0 rz 180 deg; joints [-146.495, -87.033, -23.027, 62.611, 38.441, -56.516]
  Call Extruder(654.22535)
  MoveL 2911 to (238.12, 158.03, 50.44) mm, rotated rx 180 ry 0 rz -180 deg; joints [-146.477, -87.035, -23.022, 62.63, 38.454, -56.532]
  MoveL 2912 to (238.12, 158.03, 50.44) mm, rotated rx 180 ry 0 rz -180 deg; joints [-146.477, -87.035, -23.022, 62.63, 38.454, -56.532]
  Call Extruder(654.55818)
  MoveL 2913 to (237.8, 158.48, 50.44) mm, rotated rx 180 ry 0 rz 180 deg; joints [-146.427, -87.03, -23.033, 62.668, 38.499, -56.559]
  MoveL 2914 to (237.8, 158.48, 50.44) mm, rotated rx 180 ry 0 rz 180 deg; joints [-146.427, -87.03, -23.033, 62.668, 38.499, -56.559]
  Call Extruder(654.89221)
  MoveL 2915 to (237.47, 158.93, 50.44) mm, rotated rx 180 ry 0 rz 180 deg; joints [-146.377, -87.024, -23.044, 62.706, 38.543, -56.585]
  MoveL 2916 to (237.47, 158.93, 50.44) mm, rotated rx 180 ry 0 rz 180 deg; joints [-146.377, -87.024, -23.044, 62.706, 38.543, -56.585]
  Call Extruder(655.05980)
  MoveL 2917 to (237.3, 159.15, 50.44) mm, rotated rx 180 ry 0 rz 180 deg; joints [-146.352, -87.022, -23.049, 62.725, 38.565, -56.599]
  Call Extruder(655.88912)
  MoveL 2918 to (236.39, 160.19, 50.44) mm, rotated rx 180 ry 0 rz 180 deg; joints [-146.229, -86.98, -23.134, 62.785, 38.688, -56.621]
  Call Extruder(656.52018)
  MoveL 2919 to (235.6, 160.89, 50.44) mm, rotated rx -180 ry 0 rz -180 deg; joints [-146.138, -86.92, -23.257, 62.796, 38.792, -56.595]
  MoveL 2920 to (235.6, 160.89, 50.44) mm, rotated rx -180 ry 0 rz -180 deg; joints [-146.138, -86.92, -23.257, 62.796, 38.792, -56.595]
  Call Extruder(656.71780)
  MoveL 2921 to (235.35, 161.1, 50.44) mm, rotated rx 180 ry 0 rz 180 deg; joints [-146.109, -86.9, -23.298, 62.797, 38.826, -56.585]
  Call Extruder(657.05182)
  MoveL 2922 to (234.9, 161.43, 50.44) mm, rotated rx 180 ry 0 rz -180 deg; joints [-146.062, -86.857, -23.386, 62.789, 38.886, -56.553]
  MoveL 2923 to (234.9, 161.43, 50.44) mm, rotated rx 180 ry 0 rz -180 deg; joints [-146.062, -86.857, -23.386, 62.789, 38.886, -56.553]
  Call Extruder(657.38465)
  MoveL 2924 to (234.45, 161.76, 50.44) mm, rotated rx -180 ry 0 rz 180 deg; joints [-146.015, -86.814, -23.474, 62.781, 38.945, -56.522]
  MoveL 2925 to (234.45, 161.76, 50.44) mm, rotated rx -180 ry 0 rz 180 deg; joints [-146.015, -86.814, -23.474, 62.781, 38.945, -56.522]
  Call Extruder(657.56385)
  MoveL 2926 to (234.21, 161.93, 50.44) mm, rotated rx -180 ry 0 rz 180 deg; joints [-145.99, -86.791, -23.522, 62.776, 38.978, -56.504]
  MoveL 2927 to (234.21, 161.93, 50.44) mm, rotated rx -180 ry 0 rz 180 deg; joints [-145.99, -86.791, -23.522, 62.776, 38.978, -56.504]
  Call Extruder(657.77197)
  MoveL 2928 to (233.9, 162.11, 50.44) mm, rotated rx -180 ry 0 rz 180 deg; joints [-145.961, -86.756, -23.592, 62.762, 39.018, -56.473]
  MoveL 2929 to (233.9, 162.11, 50.44) mm, rotated rx -180 ry 0 rz 180 deg; joints [-145.961, -86.756, -23.592, 62.762, 39.018, -56.473]
  Call Extruder(657.97930)
  MoveL 2930 to (233.6, 162.29, 50.44) mm, rotated rx 180 ry 0 rz -180 deg; joints [-145.933, -86.722, -23.662, 62.747, 39.058, -56.441]
  MoveL 2931 to (233.6, 162.29, 50.44) mm, rotated rx 180 ry 0 rz -180 deg; joints [-145.933, -86.722, -23.662, 62.747, 39.058, -56.441]
  Call Extruder(658.18586)
  MoveL 2932 to (233.29, 162.46, 50.44) mm, rotated rx -180 ry 0 rz -180 deg; joints [-145.905, -86.688, -23.732, 62.733, 39.098, -56.41]
  MoveL 2933 to (233.29, 162.46, 50.44) mm, rotated rx -180 ry 0 rz -180 deg; joints [-145.905, -86.688, -23.732, 62.733, 39.098, -56.41]
  Call Extruder(658.39164)
  MoveL 2934 to (232.99, 162.64, 50.44) mm, rotated rx 180 ry 0 rz -180 deg; joints [-145.876, -86.654, -23.802, 62.719, 39.138, -56.379]
  MoveL 2935 to (232.99, 162.64, 50.44) mm, rotated rx 180 ry 0 rz -180 deg; joints [-145.876, -86.654, -23.802, 62.719, 39.138, -56.379]
  Call Extruder(658.54991)
  MoveL 2936 to (232.74, 162.74, 50.44) mm, rotated rx 180 ry 0 rz -180 deg; joints [-145.856, -86.621, -23.869, 62.699, 39.171, -56.346]
  MoveL 2937 to (232.74, 162.74, 50.44) mm, rotated rx 180 ry 0 rz -180 deg; joints [-145.856, -86.621, -23.869, 62.699, 39.171, -56.346]
  Call Extruder(658.70759)
  MoveL 2938 to (232.49, 162.85, 50.44) mm, rotated rx 180 ry 0 rz 180 deg; joints [-145.835, -86.589, -23.935, 62.68, 39.203, -56.312]
  MoveL 2939 to (232.49, 162.85, 50.44) mm, rotated rx 180 ry 0 rz 180 deg; joints [-145.835, -86.589, -23.935, 62.68, 39.203, -56.312]
  Call Extruder(658.87768)
  MoveL 2940 to (232.22, 162.96, 50.44) mm, rotated rx 180 ry 0 rz 180 deg; joints [-145.813, -86.553, -24.007, 62.66, 39.239, -56.275]
  MoveL 2941 to (232.22, 162.96, 50.44) mm, rotated rx 180 ry 0 rz 180 deg; joints [-145.813, -86.553, -24.007, 62.66, 39.239, -56.275]
  Call Extruder(659.06004)
  MoveL 2942 to (231.93, 163.09, 50.44) mm, rotated rx -180 ry 0 rz 180 deg; joints [-145.789, -86.515, -24.086, 62.637, 39.277, -56.235]
  MoveL 2943 to (231.93, 163.09, 50.44) mm, rotated rx -180 ry 0 rz 180 deg; joints [-145.789, -86.515, -24.086, 62.637, 39.277, -56.235]
  Call Extruder(659.24164)
  MoveL 2944 to (231.64, 163.21, 50.44) mm, rotated rx -180 ry 0 rz 180 deg; joints [-145.766, -86.477, -24.164, 62.614, 39.315, -56.195]
  MoveL 2945 to (231.64, 163.21, 50.44) mm, rotated rx -180 ry 0 rz 180 deg; joints [-145.766, -86.477, -24.164, 62.614, 39.315, -56.195]
  Call Extruder(659.35509)
  MoveL 2946 to (231.45, 163.27, 50.44) mm, rotated rx 180 ry 0 rz -180 deg; joints [-145.751, -86.45, -24.219, 62.596, 39.34, -56.165]
  MoveL 2947 to (231.45, 163.27, 50.44) mm, rotated rx 180 ry 0 rz -180 deg; joints [-145.751, -86.45, -24.219, 62.596, 39.34, -56.165]
  Call Extruder(659.46809)
  MoveL 2948 to (231.26, 163.33, 50.44) mm, rotated rx -180 ry 0 rz 180 deg; joints [-145.737, -86.424, -24.273, 62.578, 39.364, -56.135]
  MoveL 2949 to (231.26, 163.33, 50.44) mm, rotated rx -180 ry 0 rz 180 deg; joints [-145.737, -86.424, -24.273, 62.578, 39.364, -56.135]
  Call Extruder(659.58064)
  MoveL 2950 to (231.07, 163.39, 50.44) mm, rotated rx -180 ry 0 rz 180 deg; joints [-145.723, -86.397, -24.327, 62.561, 39.389, -56.106]
  MoveL 2951 to (231.07, 163.39, 50.44) mm, rotated rx -180 ry 0 rz 180 deg; joints [-145.723, -86.397, -24.327, 62.561, 39.389, -56.106]
  Call Extruder(659.69275)
  MoveL 2952 to (230.88, 163.45, 50.44) mm, rotated rx 180 ry 0 rz -180 deg; joints [-145.709, -86.371, -24.382, 62.543, 39.414, -56.077]
  MoveL 2953 to (230.88, 163.45, 50.44) mm, rotated rx 180 ry 0 rz -180 deg; joints [-145.709, -86.371, -24.382, 62.543, 39.414, -56.077]
  Call Extruder(659.80442)
  MoveL 2954 to (230.7, 163.51, 50.44) mm, rotated rx -180 ry 0 rz -180 deg; joints [-145.695, -86.344, -24.436, 62.526, 39.438, -56.048]
  MoveL 2955 to (230.7, 163.51, 50.44) mm, rotated rx -180 ry 0 rz -180 deg; joints [-145.695, -86.344, -24.436, 62.526, 39.438, -56.048]
  Call Extruder(659.93552)
  MoveL 2956 to (230.47, 163.58, 50.44) mm, rotated rx -180 ry 0 rz 180 deg; joints [-145.679, -86.312, -24.502, 62.504, 39.467, -56.012]
  MoveL 2957 to (230.47, 163.58, 50.44) mm, rotated rx -180 ry 0 rz 180 deg; joints [-145.679, -86.312, -24.502, 62.504, 39.467, -56.012]
  Call Extruder(660.06605)
  MoveL 2958 to (230.25, 163.65, 50.44) mm, rotated rx 180 ry 0 rz 180 deg; joints [-145.662, -86.28, -24.567, 62.482, 39.496, -55.976]
  MoveL 2959 to (230.25, 163.65, 50.44) mm, rotated rx 180 ry 0 rz 180 deg; joints [-145.662, -86.28, -24.567, 62.482, 39.496, -55.976]
  Call Extruder(660.19601)
  MoveL 2960 to (230.02, 163.72, 50.44) mm, rotated rx 180 ry 0 rz 180 deg; joints [-145.646, -86.248, -24.632, 62.461, 39.525, -55.941]
  MoveL 2961 to (230.02, 163.72, 50.44) mm, rotated rx 180 ry 0 rz 180 deg; joints [-145.646, -86.248, -24.632, 62.461, 39.525, -55.941]
  Call Extruder(660.32541)
  MoveL 2962 to (229.8, 163.78, 50.44) mm, rotated rx -180 ry 0 rz 180 deg; joints [-145.629, -86.217, -24.698, 62.439, 39.554, -55.905]
  MoveL 2963 to (229.8, 163.78, 50.44) mm, rotated rx -180 ry 0 rz 180 deg; joints [-145.629, -86.217, -24.698, 62.439, 39.554, -55.905]
  Call Extruder(660.44739)
  MoveL 2964 to (229.59, 163.84, 50.44) mm, rotated rx -180 ry 0 rz 180 deg; joints [-145.614, -86.185, -24.762, 62.417, 39.582, -55.87]
  MoveL 2965 to (229.59, 163.84, 50.44) mm, rotated rx -180 ry 0 rz 180 deg; joints [-145.614, -86.185, -24.762, 62.417, 39.582, -55.87]
  Call Extruder(660.56223)
  MoveL 2966 to (229.38, 163.88, 50.44) mm, rotated rx -180 ry 0 rz 180 deg; joints [-145.601, -86.154, -24.826, 62.394, 39.608, -55.834]
  MoveL 2967 to (229.38, 163.88, 50.44) mm, rotated rx -180 ry 0 rz 180 deg; joints [-145.601, -86.154, -24.826, 62.394, 39.608, -55.834]
  Call Extruder(660.67663)
  MoveL 2968 to (229.18, 163.93, 50.44) mm, rotated rx 180 ry 0 rz -180 deg; joints [-145.587, -86.124, -24.889, 62.372, 39.635, -55.798]
  MoveL 2969 to (229.18, 163.93, 50.44) mm, rotated rx 180 ry 0 rz -180 deg; joints [-145.587, -86.124, -24.889, 62.372, 39.635, -55.798]
  Call Extruder(660.79057)
  MoveL 2970 to (228.97, 163.97, 50.44) mm, rotated rx 180 ry 0 rz 180 deg; joints [-145.573, -86.093, -24.952, 62.349, 39.661, -55.762]
  MoveL 2971 to (228.97, 163.97, 50.44) mm, rotated rx 180 ry 0 rz 180 deg; joints [-145.573, -86.093, -24.952, 62.349, 39.661, -55.762]
  Call Extruder(660.90406)
  MoveL 2972 to (228.77, 164.02, 50.44) mm, rotated rx 180 ry 0 rz 180 deg; joints [-145.559, -86.062, -25.015, 62.326, 39.688, -55.726]
  MoveL 2973 to (228.77, 164.02, 50.44) mm, rotated rx 180 ry 0 rz 180 deg; joints [-145.559, -86.062, -25.015, 62.326, 39.688, -55.726]
  Call Extruder(661.04134)
  MoveL 2974 to (228.52, 164.07, 50.44) mm, rotated rx -180 ry 0 rz 180 deg; joints [-145.543, -86.024, -25.093, 62.298, 39.72, -55.682]
  MoveL 2975 to (228.52, 164.07, 50.44) mm, rotated rx -180 ry 0 rz 180 deg; joints [-145.543, -86.024, -25.093, 62.298, 39.72, -55.682]
  Call Extruder(661.17802)
  MoveL 2976 to (228.27, 164.12, 50.44) mm, rotated rx 180 ry 0 rz 180 deg; joints [-145.527, -85.986, -25.171, 62.27, 39.752, -55.638]
  MoveL 2977 to (228.27, 164.12, 50.44) mm, rotated rx 180 ry 0 rz 180 deg; joints [-145.527, -85.986, -25.171, 62.27, 39.752, -55.638]
  Call Extruder(661.31408)
  MoveL 2978 to (228.02, 164.17, 50.44) mm, rotated rx 180 ry 0 rz -180 deg; joints [-145.51, -85.948, -25.249, 62.242, 39.784, -55.594]
  MoveL 2979 to (228.02, 164.17, 50.44) mm, rotated rx 180 ry 0 rz -180 deg; joints [-145.51, -85.948, -25.249, 62.242, 39.784, -55.594]
  Call Extruder(661.44953)
  MoveL 2980 to (227.77, 164.22, 50.44) mm, rotated rx -180 ry 0 rz -180 deg; joints [-145.494, -85.91, -25.327, 62.214, 39.816, -55.55]
  MoveL 2981 to (227.77, 164.22, 50.44) mm, rotated rx -180 ry 0 rz -180 deg; joints [-145.494, -85.91, -25.327, 62.214, 39.816, -55.55]
  Call Extruder(661.58438)
  MoveL 2982 to (227.52, 164.27, 50.44) mm, rotated rx 180 ry 0 rz -180 deg; joints [-145.477, -85.873, -25.404, 62.187, 39.848, -55.506]
  MoveL 2983 to (227.52, 164.27, 50.44) mm, rotated rx 180 ry 0 rz -180 deg; joints [-145.477, -85.873, -25.404, 62.187, 39.848, -55.506]
  Call Extruder(661.71861)
  MoveL 2984 to (227.27, 164.32, 50.44) mm, rotated rx 180 ry 0 rz 180 deg; joints [-145.461, -85.835, -25.481, 62.16, 39.88, -55.463]
  MoveL 2985 to (227.27, 164.32, 50.44) mm, rotated rx 180 ry 0 rz 180 deg; joints [-145.461, -85.835, -25.481, 62.16, 39.88, -55.463]
  Call Extruder(661.85223)
  MoveL 2986 to (227.03, 164.37, 50.44) mm, rotated rx 180 ry 0 rz -180 deg; joints [-145.444, -85.798, -25.558, 62.132, 39.913, -55.419]
  MoveL 2987 to (227.03, 164.37, 50.44) mm, rotated rx 180 ry 0 rz -180 deg; joints [-145.444, -85.798, -25.558, 62.132, 39.913, -55.419]
  Call Extruder(662.01433)
  MoveL 2988 to (226.72, 164.41, 50.44) mm, rotated rx -180 ry 0 rz 180 deg; joints [-145.425, -85.751, -25.655, 62.096, 39.952, -55.364]
  MoveL 2989 to (226.72, 164.41, 50.44) mm, rotated rx -180 ry 0 rz 180 deg; joints [-145.425, -85.751, -25.655, 62.096, 39.952, -55.364]
  Call Extruder(662.17571)
  MoveL 2990 to (226.41, 164.46, 50.44) mm, rotated rx 180 ry 0 rz 180 deg; joints [-145.406, -85.703, -25.753, 62.061, 39.991, -55.308]
  MoveL 2991 to (226.41, 164.46, 50.44) mm, rotated rx 180 ry 0 rz 180 deg; joints [-145.406, -85.703, -25.753, 62.061, 39.991, -55.308]
  Call Extruder(662.33636)
  MoveL 2992 to (226.11, 164.51, 50.44) mm, rotated rx 180 ry 0 rz 180 deg; joints [-145.386, -85.656, -25.849, 62.026, 40.03, -55.253]
  MoveL 2993 to (226.11, 164.51, 50.44) mm, rotated rx 180 ry 0 rz 180 deg; joints [-145.386, -85.656, -25.849, 62.026, 40.03, -55.253]
  Call Extruder(662.49628)
  MoveL 2994 to (225.8, 164.56, 50.44) mm, rotated rx -180 ry 0 rz 180 deg; joints [-145.367, -85.61, -25.946, 61.991, 40.069, -55.198]
  MoveL 2995 to (225.8, 164.56, 50.44) mm, rotated rx -180 ry 0 rz 180 deg; joints [-145.367, -85.61, -25.946, 61.991, 40.069, -55.198]
  Call Extruder(662.65547)
  MoveL 2996 to (225.5, 164.61, 50.44) mm, rotated rx -180 ry 0 rz 180 deg; joints [-145.348, -85.563, -26.042, 61.956, 40.109, -55.143]
  MoveL 2997 to (225.5, 164.61, 50.44) mm, rotated rx -180 ry 0 rz 180 deg; joints [-145.348, -85.563, -26.042, 61.956, 40.109, -55.143]
  Call Extruder(662.81393)
  MoveL 2998 to (225.19, 164.66, 50.44) mm, rotated rx 180 ry 0 rz 180 deg; joints [-145.328, -85.516, -26.138, 61.921, 40.148, -55.088]
  MoveL 2999 to (225.19, 164.66, 50.44) mm, rotated rx 180 ry 0 rz 180 deg; joints [-145.328, -85.516, -26.138, 61.921, 40.148, -55.088]
  Call Extruder(663.01281)
  MoveL 3000 to (224.8, 164.7, 50.44) mm, rotated rx 180 ry 0 rz 180 deg; joints [-145.305, -85.456, -26.263, 61.875, 40.197, -55.016]
  MoveL 3001 to (224.8, 164.7, 50.44) mm, rotated rx 180 ry 0 rz 180 deg; joints [-145.305, -85.456, -26.263, 61.875, 40.197, -55.016]
  Call Extruder(663.21082)
  MoveL 3002 to (224.42, 164.75, 50.44) mm, rotated rx 180 ry 0 rz 180 deg; joints [-145.281, -85.395, -26.388, 61.829, 40.247, -54.945]
  MoveL 3003 to (224.42, 164.75, 50.44) mm, rotated rx 180 ry 0 rz 180 deg; joints [-145.281, -85.395, -26.388, 61.829, 40.247, -54.945]
  Call Extruder(663.40796)
  MoveL 3004 to (224.03, 164.79, 50.44) mm, rotated rx -180 ry 0 rz 180 deg; joints [-145.258, -85.335, -26.512, 61.783, 40.296, -54.873]
  MoveL 3005 to (224.03, 164.79, 50.44) mm, rotated rx -180 ry 0 rz 180 deg; joints [-145.258, -85.335, -26.512, 61.783, 40.296, -54.873]
  Call Extruder(663.60423)
  MoveL 3006 to (223.64, 164.84, 50.44) mm, rotated rx -180 ry 0 rz 180 deg; joints [-145.234, -85.275, -26.636, 61.738, 40.346, -54.802]
  MoveL 3007 to (223.64, 164.84, 50.44) mm, rotated rx -180 ry 0 rz 180 deg; joints [-145.234, -85.275, -26.636, 61.738, 40.346, -54.802]
  Call Extruder(663.84990)
  MoveL 3008 to (223.15, 164.89, 50.44) mm, rotated rx -180 ry 0 rz 180 deg; joints [-145.206, -85.198, -26.794, 61.679, 40.408, -54.711]
  MoveL 3009 to (223.15, 164.89, 50.44) mm, rotated rx -180 ry 0 rz 180 deg; joints [-145.206, -85.198, -26.794, 61.679, 40.408, -54.711]
  Call Extruder(664.14459)
  MoveL 3010 to (222.56, 164.93, 50.44) mm, rotated rx -180 ry 0 rz 180 deg; joints [-145.172, -85.105, -26.986, 61.607, 40.483, -54.6]
  MoveL 3011 to (222.56, 164.93, 50.44) mm, rotated rx -180 ry 0 rz 180 deg; joints [-145.172, -85.105, -26.986, 61.607, 40.483, -54.6]
  Call Extruder(664.43795)
  MoveL 3012 to (221.97, 164.98, 50.44) mm, rotated rx 180 ry 0 rz 180 deg; joints [-145.138, -85.012, -27.177, 61.536, 40.557, -54.489]
  MoveL 3013 to (221.97, 164.98, 50.44) mm, rotated rx 180 ry 0 rz 180 deg; joints [-145.138, -85.012, -27.177, 61.536, 40.557, -54.489]
  Call Extruder(664.87126)
  MoveL 3014 to (221.1, 165.02, 50.44) mm, rotated rx 180 ry 0 rz 180 deg; joints [-145.088, -84.873, -27.465, 61.428, 40.668, -54.322]
  MoveL 3015 to (221.1, 165.02, 50.44) mm, rotated rx 180 ry 0 rz 180 deg; joints [-145.088, -84.873, -27.465, 61.428, 40.668, -54.322]
  Call Extruder(665.44342)
  MoveL 3016 to (219.94, 165.07, 50.44) mm, rotated rx 180 ry 0 rz -180 deg; joints [-145.024, -84.688, -27.847, 61.284, 40.815, -54.1]
  MoveL 3017 to (219.94, 165.07, 50.44) mm, rotated rx 180 ry 0 rz -180 deg; joints [-145.024, -84.688, -27.847, 61.284, 40.815, -54.1]
  Call Extruder(665.87130)
  MoveL 3018 to (219.06, 165.09, 50.44) mm, rotated rx 180 ry 0 rz -180 deg; joints [-144.977, -84.549, -28.136, 61.175, 40.925, -53.932]
  Call Extruder(782.51995)
  MoveL 3019 to (-19.06, 165.09, 50.44) mm, rotated rx -180 ry 0 rz 180 deg; joints [-127.435, -64.173, -74.502, 60.106, 66.335, -34.923]
  MoveL 3020 to (-19.06, 165.09, 50.44) mm, rotated rx -180 ry 0 rz 180 deg; joints [-127.435, -64.173, -74.502, 60.106, 66.335, -34.923]
  Call Extruder(783.23557)
  MoveL 3021 to (-20.52, 165.05, 50.44) mm, rotated rx 180 ry 0 rz 180 deg; joints [-127.291, -64.104, -74.685, 60.191, 66.474, -34.867]
  MoveL 3022 to (-20.52, 165.05, 50.44) mm, rotated rx 180 ry 0 rz 180 deg; joints [-127.291, -64.104, -74.685, 60.191, 66.474, -34.867]
  Call Extruder(783.81031)
  MoveL 3023 to (-21.68, 165, 50.44) mm, rotated rx -180 ry 0 rz 180 deg; joints [-127.178, -64.048, -74.833, 60.258, 66.585, -34.82]
  MoveL 3024 to (-21.68, 165, 50.44) mm, rotated rx -180 ry 0 rz 180 deg; joints [-127.178, -64.048, -74.833, 60.258, 66.585, -34.82]
  Call Extruder(784.10367)
  MoveL 3025 to (-22.27, 164.95, 50.44) mm, rotated rx 180 ry 0 rz 180 deg; joints [-127.122, -64.019, -74.911, 60.29, 66.641, -34.794]
  MoveL 3026 to (-22.27, 164.95, 50.44) mm, rotated rx 180 ry 0 rz 180 deg; joints [-127.122, -64.019, -74.911, 60.29, 66.641, -34.794]
  Call Extruder(784.39837)
  MoveL 3027 to (-22.86, 164.91, 50.44) mm, rotated rx -180 ry 0 rz 180 deg; joints [-127.065, -63.989, -74.989, 60.322, 66.697, -34.768]
  MoveL 3028 to (-22.86, 164.91, 50.44) mm, rotated rx -180 ry 0 rz 180 deg; joints [-127.065, -63.989, -74.989, 60.322, 66.697, -34.768]
  Call Extruder(784.69439)
  MoveL 3029 to (-23.45, 164.86, 50.44) mm, rotated rx 180 ry 0 rz 180 deg; joints [-127.009, -63.96, -75.067, 60.354, 66.753, -34.741]
  MoveL 3030 to (-23.45, 164.86, 50.44) mm, rotated rx 180 ry 0 rz 180 deg; joints [-127.009, -63.96, -75.067, 60.354, 66.753, -34.741]
  Call Extruder(784.89067)
  MoveL 3031 to (-23.83, 164.82, 50.44) mm, rotated rx 180 ry 0 rz -180 deg; joints [-126.973, -63.94, -75.121, 60.374, 66.79, -34.722]
  MoveL 3032 to (-23.83, 164.82, 50.44) mm, rotated rx 180 ry 0 rz -180 deg; joints [-126.973, -63.94, -75.121, 60.374, 66.79, -34.722]
  Call Extruder(785.08781)
  MoveL 3033 to (-24.22, 164.77, 50.44) mm, rotated rx -180 ry 0 rz 180 deg; joints [-126.937, -63.919, -75.174, 60.393, 66.827, -34.703]
  MoveL 3034 to (-24.22, 164.77, 50.44) mm, rotated rx -180 ry 0 rz 180 deg; joints [-126.937, -63.919, -75.174, 60.393, 66.827, -34.703]
  Call Extruder(785.28582)
  MoveL 3035 to (-24.61, 164.72, 50.44) mm, rotated rx 180 ry 0 rz 180 deg; joints [-126.901, -63.899, -75.228, 60.413, 66.864, -34.684]
  MoveL 3036 to (-24.61, 164.72, 50.44) mm, rotated rx 180 ry 0 rz 180 deg; joints [-126.901, -63.899, -75.228, 60.413, 66.864, -34.684]
  Call Extruder(785.48469)
  MoveL 3037 to (-25, 164.68, 50.44) mm, rotated rx 180 ry 0 rz 180 deg; joints [-126.865, -63.879, -75.282, 60.433, 66.901, -34.665]
  MoveL 3038 to (-25, 164.68, 50.44) mm, rotated rx 180 ry 0 rz 180 deg; joints [-126.865, -63.879, -75.282, 60.433, 66.901, -34.665]
  Call Extruder(785.66377)
  MoveL 3039 to (-25.34, 164.63, 50.44) mm, rotated rx -180 ry 0 rz -180 deg; joints [-126.834, -63.861, -75.33, 60.45, 66.934, -34.648]
  MoveL 3040 to (-25.34, 164.63, 50.44) mm, rotated rx -180 ry 0 rz -180 deg; joints [-126.834, -63.861, -75.33, 60.45, 66.934, -34.648]
  Call Extruder(785.82297)
  MoveL 3041 to (-25.65, 164.58, 50.44) mm, rotated rx 180 ry 0 rz 180 deg; joints [-126.806, -63.844, -75.374, 60.464, 66.963, -34.631]
  MoveL 3042 to (-25.65, 164.58, 50.44) mm, rotated rx 180 ry 0 rz 180 deg; joints [-126.806, -63.844, -75.374, 60.464, 66.963, -34.631]
  Call Extruder(785.98289)
  MoveL 3043 to (-25.96, 164.54, 50.44) mm, rotated rx -180 ry 0 rz 180 deg; joints [-126.779, -63.828, -75.418, 60.479, 66.993, -34.615]
  MoveL 3044 to (-25.96, 164.54, 50.44) mm, rotated rx -180 ry 0 rz 180 deg; joints [-126.779, -63.828, -75.418, 60.479, 66.993, -34.615]
  Call Extruder(786.14354)
  MoveL 3045 to (-26.26, 164.49, 50.44) mm, rotated rx 180 ry 0 rz 180 deg; joints [-126.751, -63.811, -75.462, 60.493, 67.022, -34.598]
  MoveL 3046 to (-26.26, 164.49, 50.44) mm, rotated rx 180 ry 0 rz 180 deg; joints [-126.751, -63.811, -75.462, 60.493, 67.022, -34.598]
  Call Extruder(786.30492)
  MoveL 3047 to (-26.57, 164.44, 50.44) mm, rotated rx -180 ry 0 rz 180 deg; joints [-126.723, -63.795, -75.506, 60.508, 67.051, -34.582]
  MoveL 3048 to (-26.57, 164.44, 50.44) mm, rotated rx -180 ry 0 rz 180 deg; joints [-126.723, -63.795, -75.506, 60.508, 67.051, -34.582]
  Call Extruder(786.46703)
  MoveL 3049 to (-26.87, 164.39, 50.44) mm, rotated rx 180 ry 0 rz 180 deg; joints [-126.696, -63.779, -75.55, 60.522, 67.08, -34.566]
  MoveL 3050 to (-26.87, 164.39, 50.44) mm, rotated rx 180 ry 0 rz 180 deg; joints [-126.696, -63.779, -75.55, 60.522, 67.08, -34.566]
  Call Extruder(786.61523)
  MoveL 3051 to (-27.15, 164.34, 50.44) mm, rotated rx -180 ry 0 rz 180 deg; joints [-126.671, -63.763, -75.591, 60.535, 67.107, -34.55]
  MoveL 3052 to (-27.15, 164.34, 50.44) mm, rotated rx -180 ry 0 rz 180 deg; joints [-126.671, -63.763, -75.591, 60.535, 67.107, -34.55]
  Call Extruder(786.74946)
  MoveL 3053 to (-27.4, 164.29, 50.44) mm, rotated rx 180 ry 0 rz 180 deg; joints [-126.649, -63.75, -75.628, 60.546, 67.13, -34.536]
  MoveL 3054 to (-27.4, 164.29, 50.44) mm, rotated rx 180 ry 0 rz 180 deg; joints [-126.649, -63.75, -75.628, 60.546, 67.13, -34.536]
  Call Extruder(786.88430)
  MoveL 3055 to (-27.65, 164.24, 50.44) mm, rotated rx 180 ry 0 rz 180 deg; joints [-126.628, -63.736, -75.665, 60.557, 67.154, -34.521]
  MoveL 3056 to (-27.65, 164.24, 50.44) mm, rotated rx 180 ry 0 rz 180 deg; joints [-126.628, -63.736, -75.665, 60.557, 67.154, -34.521]
  Call Extruder(787.01975)
  MoveL 3057 to (-27.9, 164.19, 50.44) mm, rotated rx 180 ry 0 rz 180 deg; joints [-126.606, -63.722, -75.703, 60.568, 67.178, -34.507]
  MoveL 3058 to (-27.9, 164.19, 50.44) mm, rotated rx 180 ry 0 rz 180 deg; joints [-126.606, -63.722, -75.703, 60.568, 67.178, -34.507]
  Call Extruder(787.15582)
  MoveL 3059 to (-28.15, 164.14, 50.44) mm, rotated rx 180 ry 0 rz 180 deg; joints [-126.584, -63.708, -75.74, 60.579, 67.202, -34.492]
  MoveL 3060 to (-28.15, 164.14, 50.44) mm, rotated rx 180 ry 0 rz 180 deg; joints [-126.584, -63.708, -75.74, 60.579, 67.202, -34.492]
  Call Extruder(787.29249)
  MoveL 3061 to (-28.4, 164.09, 50.44) mm, rotated rx 180 ry 0 rz 180 deg; joints [-126.562, -63.694, -75.777, 60.59, 67.226, -34.478]
  MoveL 3062 to (-28.4, 164.09, 50.44) mm, rotated rx 180 ry 0 rz 180 deg; joints [-126.562, -63.694, -75.777, 60.59, 67.226, -34.478]
  Call Extruder(787.42977)
  MoveL 3063 to (-28.65, 164.04, 50.44) mm, rotated rx -180 ry 0 rz 180 deg; joints [-126.54, -63.68, -75.814, 60.601, 67.25, -34.463]
  MoveL 3064 to (-28.65, 164.04, 50.44) mm, rotated rx -180 ry 0 rz 180 deg; joints [-126.54, -63.68, -75.814, 60.601, 67.25, -34.463]
  Call Extruder(787.55544)
  MoveL 3065 to (-28.87, 164, 50.44) mm, rotated rx -180 ry 0 rz 180 deg; joints [-126.52, -63.667, -75.848, 60.611, 67.271, -34.45]
  MoveL 3066 to (-28.87, 164, 50.44) mm, rotated rx -180 ry 0 rz 180 deg; joints [-126.52, -63.667, -75.848, 60.611, 67.271, -34.45]
  Call Extruder(787.66938)
  MoveL 3067 to (-29.08, 163.95, 50.44) mm, rotated rx 180 ry 0 rz -180 deg; joints [-126.503, -63.656, -75.88, 60.62, 67.291, -34.438]
  MoveL 3068 to (-29.08, 163.95, 50.44) mm, rotated rx 180 ry 0 rz -180 deg; joints [-126.503, -63.656, -75.88, 60.62, 67.291, -34.438]
  Call Extruder(787.78378)
  MoveL 3069 to (-29.28, 163.91, 50.44) mm, rotated rx 180 ry 0 rz 180 deg; joints [-126.485, -63.644, -75.91, 60.628, 67.31, -34.425]
  MoveL 3070 to (-29.28, 163.91, 50.44) mm, rotated rx 180 ry 0 rz 180 deg; joints [-126.485, -63.644, -75.91, 60.628, 67.31, -34.425]
  Call Extruder(787.89862)
  MoveL 3071 to (-29.48, 163.86, 50.44) mm, rotated rx 180 ry 0 rz -180 deg; joints [-126.467, -63.633, -75.942, 60.637, 67.33, -34.413]
  MoveL 3072 to (-29.48, 163.86, 50.44) mm, rotated rx 180 ry 0 rz -180 deg; joints [-126.467, -63.633, -75.942, 60.637, 67.33, -34.413]
  Call Extruder(788.01392)
  MoveL 3073 to (-29.69, 163.82, 50.44) mm, rotated rx 180 ry 0 rz 180 deg; joints [-126.45, -63.621, -75.973, 60.646, 67.349, -34.401]
  MoveL 3074 to (-29.69, 163.82, 50.44) mm, rotated rx 180 ry 0 rz 180 deg; joints [-126.45, -63.621, -75.973, 60.646, 67.349, -34.401]
  Call Extruder(788.14332)
  MoveL 3075 to (-29.91, 163.75, 50.44) mm, rotated rx -180 ry 0 rz 180 deg; joints [-126.432, -63.607, -76.009, 60.653, 67.371, -34.385]
  MoveL 3076 to (-29.91, 163.75, 50.44) mm, rotated rx -180 ry 0 rz 180 deg; joints [-126.432, -63.607, -76.009, 60.653, 67.371, -34.385]
  Call Extruder(788.27328)
  MoveL 3077 to (-30.14, 163.68, 50.44) mm, rotated rx -180 ry 0 rz 180 deg; joints [-126.414, -63.594, -76.046, 60.661, 67.392, -34.369]
  MoveL 3078 to (-30.14, 163.68, 50.44) mm, rotated rx -180 ry 0 rz 180 deg; joints [-126.414, -63.594, -76.046, 60.661, 67.392, -34.369]
  Call Extruder(788.40380)
  MoveL 3079 to (-30.36, 163.61, 50.44) mm, rotated rx 180 ry 0 rz 180 deg; joints [-126.396, -63.58, -76.083, 60.669, 67.414, -34.354]
  MoveL 3080 to (-30.36, 163.61, 50.44) mm, rotated rx 180 ry 0 rz 180 deg; joints [-126.396, -63.58, -76.083, 60.669, 67.414, -34.354]
  Call Extruder(788.53489)
  MoveL 3081 to (-30.58, 163.55, 50.44) mm, rotated rx 180 ry 0 rz 180 deg; joints [-126.378, -63.566, -76.12, 60.676, 67.435, -34.338]
  MoveL 3082 to (-30.58, 163.55, 50.44) mm, rotated rx 180 ry 0 rz 180 deg; joints [-126.378, -63.566, -76.12, 60.676, 67.435, -34.338]
  Call Extruder(788.65654)
  MoveL 3083 to (-30.79, 163.48, 50.44) mm, rotated rx 180 ry 0 rz 180 deg; joints [-126.361, -63.553, -76.154, 60.683, 67.455, -34.323]
  MoveL 3084 to (-30.79, 163.48, 50.44) mm, rotated rx 180 ry 0 rz 180 deg; joints [-126.361, -63.553, -76.154, 60.683, 67.455, -34.323]
  Call Extruder(788.76865)
  MoveL 3085 to (-30.98, 163.42, 50.44) mm, rotated rx -180 ry 0 rz 180 deg; joints [-126.347, -63.542, -76.186, 60.689, 67.473, -34.31]
  MoveL 3086 to (-30.98, 163.42, 50.44) mm, rotated rx -180 ry 0 rz 180 deg; joints [-126.347, -63.542, -76.186, 60.689, 67.473, -34.31]
  Call Extruder(788.88121)
  MoveL 3087 to (-31.17, 163.36, 50.44) mm, rotated rx 180 ry 0 rz 180 deg; joints [-126.332, -63.53, -76.218, 60.695, 67.492, -34.296]
  MoveL 3088 to (-31.17, 163.36, 50.44) mm, rotated rx 180 ry 0 rz 180 deg; joints [-126.332, -63.53, -76.218, 60.695, 67.492, -34.296]
  Call Extruder(788.99421)
  MoveL 3089 to (-31.35, 163.3, 50.44) mm, rotated rx 180 ry 0 rz 180 deg; joints [-126.317, -63.518, -76.249, 60.702, 67.51, -34.282]
  MoveL 3090 to (-31.35, 163.3, 50.44) mm, rotated rx 180 ry 0 rz 180 deg; joints [-126.317, -63.518, -76.249, 60.702, 67.51, -34.282]
  Call Extruder(789.10766)
  MoveL 3091 to (-31.54, 163.24, 50.44) mm, rotated rx -180 ry 0 rz 180 deg; joints [-126.302, -63.506, -76.281, 60.708, 67.528, -34.269]
  MoveL 3092 to (-31.54, 163.24, 50.44) mm, rotated rx -180 ry 0 rz 180 deg; joints [-126.302, -63.506, -76.281, 60.708, 67.528, -34.269]
  Call Extruder(789.25531)
  MoveL 3093 to (-31.78, 163.15, 50.44) mm, rotated rx 180 ry 0 rz -180 deg; joints [-126.284, -63.491, -76.323, 60.714, 67.551, -34.25]
  MoveL 3094 to (-31.78, 163.15, 50.44) mm, rotated rx 180 ry 0 rz -180 deg; joints [-126.284, -63.491, -76.323, 60.714, 67.551, -34.25]
  Call Extruder(789.43766)
  MoveL 3095 to (-32.08, 163.03, 50.44) mm, rotated rx -180 ry 0 rz -180 deg; joints [-126.263, -63.471, -76.377, 60.721, 67.579, -34.225]
  MoveL 3096 to (-32.08, 163.03, 50.44) mm, rotated rx -180 ry 0 rz -180 deg; joints [-126.263, -63.471, -76.377, 60.721, 67.579, -34.225]
  Call Extruder(789.62078)
  MoveL 3097 to (-32.37, 162.91, 50.44) mm, rotated rx 180 ry 0 rz 180 deg; joints [-126.241, -63.451, -76.429, 60.728, 67.607, -34.201]
  MoveL 3098 to (-32.37, 162.91, 50.44) mm, rotated rx 180 ry 0 rz 180 deg; joints [-126.241, -63.451, -76.429, 60.728, 67.607, -34.201]
  Call Extruder(789.77845)
  MoveL 3099 to (-32.62, 162.8, 50.44) mm, rotated rx 180 ry 0 rz 180 deg; joints [-126.224, -63.434, -76.475, 60.734, 67.631, -34.18]
  MoveL 3100 to (-32.62, 162.8, 50.44) mm, rotated rx 180 ry 0 rz 180 deg; joints [-126.224, -63.434, -76.475, 60.734, 67.631, -34.18]
  Call Extruder(789.93673)
  MoveL 3101 to (-32.86, 162.69, 50.44) mm, rotated rx -180 ry 0 rz -180 deg; joints [-126.206, -63.417, -76.521, 60.739, 67.656, -34.159]
  MoveL 3102 to (-32.86, 162.69, 50.44) mm, rotated rx -180 ry 0 rz -180 deg; joints [-126.206, -63.417, -76.521, 60.739, 67.656, -34.159]
  Call Extruder(790.11874)
  MoveL 3103 to (-33.14, 162.55, 50.44) mm, rotated rx 180 ry 0 rz -180 deg; joints [-126.188, -63.397, -76.576, 60.743, 67.683, -34.133]
  MoveL 3104 to (-33.14, 162.55, 50.44) mm, rotated rx 180 ry 0 rz -180 deg; joints [-126.188, -63.397, -76.576, 60.743, 67.683, -34.133]
  Call Extruder(790.32530)
  MoveL 3105 to (-33.45, 162.37, 50.44) mm, rotated rx 180 ry 0 rz -180 deg; joints [-126.169, -63.374, -76.638, 60.745, 67.712, -34.101]
  MoveL 3106 to (-33.45, 162.37, 50.44) mm, rotated rx 180 ry 0 rz -180 deg; joints [-126.169, -63.374, -76.638, 60.745, 67.712, -34.101]
  Call Extruder(790.53263)
  MoveL 3107 to (-33.75, 162.2, 50.44) mm, rotated rx 180 ry 0 rz 180 deg; joints [-126.151, -63.351, -76.701, 60.748, 67.742, -34.07]
  MoveL 3108 to (-33.75, 162.2, 50.44) mm, rotated rx 180 ry 0 rz 180 deg; joints [-126.151, -63.351, -76.701, 60.748, 67.742, -34.07]
  Call Extruder(790.74074)
  MoveL 3109 to (-34.05, 162.02, 50.44) mm, rotated rx 180 ry 0 rz 180 deg; joints [-126.133, -63.328, -76.764, 60.75, 67.772, -34.039]
  MoveL 3110 to (-34.05, 162.02, 50.44) mm, rotated rx 180 ry 0 rz 180 deg; joints [-126.133, -63.328, -76.764, 60.75, 67.772, -34.039]
  Call Extruder(790.85846)
  MoveL 3111 to (-34.23, 161.92, 50.44) mm, rotated rx -180 ry 0 rz 180 deg; joints [-126.122, -63.315, -76.799, 60.751, 67.788, -34.022]
  MoveL 3112 to (-34.23, 161.92, 50.44) mm, rotated rx -180 ry 0 rz 180 deg; joints [-126.122, -63.315, -76.799, 60.751, 67.788, -34.022]
  Call Extruder(791.19129)
  MoveL 3113 to (-34.68, 161.59, 50.44) mm, rotated rx -180 ry 0 rz 180 deg; joints [-126.1, -63.276, -76.903, 60.748, 67.833, -33.967]
  MoveL 3114 to (-34.68, 161.59, 50.44) mm, rotated rx -180 ry 0 rz 180 deg; joints [-126.1, -63.276, -76.903, 60.748, 67.833, -33.967]
  Call Extruder(791.52530)
  MoveL 3115 to (-35.13, 161.27, 50.44) mm, rotated rx -180 ry 0 rz 180 deg; joints [-126.078, -63.238, -77.007, 60.744, 67.877, -33.913]
  MoveL 3116 to (-35.13, 161.27, 50.44) mm, rotated rx -180 ry 0 rz 180 deg; joints [-126.078, -63.238, -77.007, 60.744, 67.877, -33.913]
  Call Extruder(791.69289)
  MoveL 3117 to (-35.35, 161.1, 50.44) mm, rotated rx 180 ry 0 rz 180 deg; joints [-126.067, -63.219, -77.059, 60.743, 67.899, -33.886]
  Call Extruder(792.52220)
  MoveL 3118 to (-36.39, 160.19, 50.44) mm, rotated rx 180 ry 0 rz 180 deg; joints [-126.027, -63.123, -77.321, 60.719, 68.002, -33.743]
  Call Extruder(793.04443)
  MoveL 3119 to (-36.97, 159.54, 50.44) mm, rotated rx 180 ry 0 rz 180 deg; joints [-126.016, -63.061, -77.489, 60.692, 68.061, -33.647]
  Set speed (130.0 mm/s)
  MoveL 3120 to (-38.97, 156.78, 50.44) mm, rotated rx 180 ry 0 rz 180 deg; joints [-126.016, -62.82, -78.149, 60.546, 68.266, -33.253]
  MoveL 3121 to (-38.97, 156.78, 59.84) mm, rotated rx 180 ry 0 rz -180 deg; joints [-126.016, -61.503, -78.86, 60.758, 67.969, -33.823]
  Call Extruder(791.04443)
  Set speed (40.0 mm/s)
  MoveL 3122 to (-38.97, 156.78, 59.84) mm, rotated rx 180 ry 0 rz -180 deg; joints [-126.016, -61.503, -78.86, 60.758, 67.969, -33.823]
  Call Extruder(0.00000)
  Set speed (130.0 mm/s)
  MoveL 3123 to (-31.64, 163.21, 59.84) mm, rotated rx 180 ry 0 rz -180 deg; joints [-126.294, -62.197, -77.008, 60.926, 67.248, -34.822]
  Call Extruder(2.00000)
  Set speed (40.0 mm/s)
  MoveL 3124 to (-31.64, 163.21, 59.84) mm, rotated rx 180 ry 0 rz -180 deg; joints [-126.294, -62.197, -77.008, 60.926, 67.248, -34.822]
  Set speed (30.0 mm/s)
  MoveL 3125 to (-31.64, 163.21, 59.84) mm, rotated rx 180 ry 0 rz -180 deg; joints [-126.294, -62.197, -77.008, 60.926, 67.248, -34.822]
  Call Extruder(2.18198)
  MoveL 3126 to (-31.93, 163.09, 59.84) mm, rotated rx 180 ry 0 rz 180 deg; joints [-126.273, -62.176, -77.061, 60.933, 67.276, -34.798]
  MoveL 3127 to (-31.93, 163.09, 59.84) mm, rotated rx 180 ry 0 rz 180 deg; joints [-126.273, -62.176, -77.061, 60.933, 67.276, -34.798]
  Call Extruder(2.36471)
  MoveL 3128 to (-32.22, 162.96, 59.84) mm, rotated rx 180 ry 0 rz 180 deg; joints [-126.252, -62.156, -77.114, 60.94, 67.304, -34.774]
  MoveL 3129 to (-32.22, 162.96, 59.84) mm, rotated rx 180 ry 0 rz 180 deg; joints [-126.252, -62.156, -77.114, 60.94, 67.304, -34.774]
  Call Extruder(2.53513)
  MoveL 3130 to (-32.49, 162.85, 59.84) mm, rotated rx 180 ry 0 rz 180 deg; joints [-126.233, -62.138, -77.164, 60.946, 67.33, -34.752]
  MoveL 3131 to (-32.49, 162.85, 59.84) mm, rotated rx 180 ry 0 rz 180 deg; joints [-126.233, -62.138, -77.164, 60.946, 67.33, -34.752]
  Call Extruder(2.69310)
  MoveL 3132 to (-32.74, 162.74, 59.84) mm, rotated rx 180 ry 0 rz 180 deg; joints [-126.215, -62.12, -77.209, 60.951, 67.354, -34.731]
  MoveL 3133 to (-32.74, 162.74, 59.84) mm, rotated rx 180 ry 0 rz 180 deg; joints [-126.215, -62.12, -77.209, 60.951, 67.354, -34.731]
  Call Extruder(2.85168)
  MoveL 3134 to (-32.99, 162.64, 59.84) mm, rotated rx -180 ry 0 rz 180 deg; joints [-126.197, -62.103, -77.255, 60.957, 67.378, -34.71]
  MoveL 3135 to (-32.99, 162.64, 59.84) mm, rotated rx -180 ry 0 rz 180 deg; joints [-126.197, -62.103, -77.255, 60.957, 67.378, -34.71]
  Call Extruder(3.05785)
  MoveL 3136 to (-33.29, 162.46, 59.84) mm, rotated rx 180 ry 0 rz 180 deg; joints [-126.179, -62.079, -77.318, 60.959, 67.408, -34.679]
  MoveL 3137 to (-33.29, 162.46, 59.84) mm, rotated rx 180 ry 0 rz 180 deg; joints [-126.179, -62.079, -77.318, 60.959, 67.408, -34.679]
  Call Extruder(3.26479)
  MoveL 3138 to (-33.6, 162.29, 59.84) mm, rotated rx -180 ry 0 rz 180 deg; joints [-126.16, -62.056, -77.381, 60.961, 67.437, -34.648]
  MoveL 3139 to (-33.6, 162.29, 59.84) mm, rotated rx -180 ry 0 rz 180 deg; joints [-126.16, -62.056, -77.381, 60.961, 67.437, -34.648]
  Call Extruder(3.47251)
  MoveL 3140 to (-33.9, 162.11, 59.84) mm, rotated rx -180 ry 0 rz 180 deg; joints [-126.142, -62.032, -77.444, 60.963, 67.466, -34.618]
  MoveL 3141 to (-33.9, 162.11, 59.84) mm, rotated rx -180 ry 0 rz 180 deg; joints [-126.142, -62.032, -77.444, 60.963, 67.466, -34.618]
  Call Extruder(3.68101)
  MoveL 3142 to (-34.21, 161.94, 59.84) mm, rotated rx -180 ry 0 rz 180 deg; joints [-126.123, -62.008, -77.507, 60.965, 67.496, -34.587]
  MoveL 3143 to (-34.21, 161.94, 59.84) mm, rotated rx -180 ry 0 rz 180 deg; joints [-126.123, -62.008, -77.507, 60.965, 67.496, -34.587]
  Call Extruder(3.86055)
  MoveL 3144 to (-34.45, 161.76, 59.84) mm, rotated rx 180 ry 0 rz 180 deg; joints [-126.111, -61.987, -77.563, 60.964, 67.52, -34.558]
  MoveL 3145 to (-34.45, 161.76, 59.84) mm, rotated rx 180 ry 0 rz 180 deg; joints [-126.111, -61.987, -77.563, 60.964, 67.52, -34.558]
  Call Extruder(4.19399)
  MoveL 3146 to (-34.9, 161.43, 59.84) mm, rotated rx 180 ry 0 rz 180 deg; joints [-126.089, -61.948, -77.666, 60.96, 67.564, -34.504]
  MoveL 3147 to (-34.9, 161.43, 59.84) mm, rotated rx 180 ry 0 rz 180 deg; joints [-126.089, -61.948, -77.666, 60.96, 67.564, -34.504]
  Call Extruder(4.52861)
  MoveL 3148 to (-35.35, 161.1, 59.84) mm, rotated rx -180 ry 0 rz 180 deg; joints [-126.067, -61.909, -77.77, 60.957, 67.608, -34.451]
  Call Extruder(5.35652)
  MoveL 3149 to (-36.39, 160.19, 59.84) mm, rotated rx -180 ry 0 rz 180 deg; joints [-126.027, -61.811, -78.032, 60.933, 67.71, -34.309]
  Call Extruder(6.18445)
  MoveL 3150 to (-37.3, 159.15, 59.84) mm, rotated rx -180 ry 0 rz 180 deg; joints [-126.011, -61.711, -78.3, 60.888, 67.801, -34.157]
  Call Extruder(6.35176)
  MoveL 3151 to (-37.47, 158.93, 59.84) mm, rotated rx 180 ry 0 rz -180 deg; joints [-126.011, -61.691, -78.354, 60.876, 67.817, -34.125]
  MoveL 3152 to (-37.47, 158.93, 59.84) mm, rotated rx 180 ry 0 rz -180 deg; joints [-126.011, -61.691, -78.354, 60.876, 67.817, -34.125]
  Call Extruder(6.68519)
  MoveL 3153 to (-37.79, 158.48, 59.84) mm, rotated rx 180 ry 0 rz 180 deg; joints [-126.011, -61.651, -78.462, 60.852, 67.85, -34.061]
  MoveL 3154 to (-37.79, 158.48, 59.84) mm, rotated rx 180 ry 0 rz 180 deg; joints [-126.011, -61.651, -78.462, 60.852, 67.85, -34.061]
  Call Extruder(7.01744)
  MoveL 3155 to (-38.12, 158.03, 59.84) mm, rotated rx 180 ry 0 rz 180 deg; joints [-126.011, -61.61, -78.57, 60.828, 67.883, -33.997]
  MoveL 3156 to (-38.12, 158.03, 59.84) mm, rotated rx 180 ry 0 rz 180 deg; joints [-126.011, -61.61, -78.57, 60.828, 67.883, -33.997]
  Call Extruder(7.13511)
  MoveL 3157 to (-38.22, 157.85, 59.84) mm, rotated rx -180 ry 0 rz 180 deg; joints [-126.013, -61.596, -78.608, 60.817, 67.893, -33.973]
  MoveL 3158 to (-38.22, 157.85, 59.84) mm, rotated rx -180 ry 0 rz 180 deg; joints [-126.013, -61.596, -78.608, 60.817, 67.893, -33.973]
  Call Extruder(7.34283)
  MoveL 3159 to (-38.4, 157.55, 59.84) mm, rotated rx 180 ry 0 rz 180 deg; joints [-126.018, -61.571, -78.676, 60.797, 67.911, -33.932]
  MoveL 3160 to (-38.4, 157.55, 59.84) mm, rotated rx 180 ry 0 rz 180 deg; joints [-126.018, -61.571, -78.676, 60.797, 67.911, -33.932]
  Call Extruder(7.54978)
  MoveL 3161 to (-38.57, 157.25, 59.84) mm, rotated rx 180 ry 0 rz 180 deg; joints [-126.023, -61.546, -78.743, 60.778, 67.929, -33.89]
  MoveL 3162 to (-38.57, 157.25, 59.84) mm, rotated rx 180 ry 0 rz 180 deg; joints [-126.023, -61.546, -78.743, 60.778, 67.929, -33.89]
  Call Extruder(7.75595)
  MoveL 3163 to (-38.75, 156.94, 59.84) mm, rotated rx -180 ry 0 rz 180 deg; joints [-126.028, -61.521, -78.81, 60.759, 67.947, -33.849]
  MoveL 3164 to (-38.75, 156.94, 59.84) mm, rotated rx -180 ry 0 rz 180 deg; joints [-126.028, -61.521, -78.81, 60.759, 67.947, -33.849]
  Call Extruder(7.93763)
  MoveL 3165 to (-38.89, 156.67, 59.84) mm, rotated rx 180 ry 0 rz -180 deg; joints [-126.034, -61.499, -78.87, 60.74, 67.962, -33.811]
  MoveL 3166 to (-38.89, 156.67, 59.84) mm, rotated rx 180 ry 0 rz -180 deg; joints [-126.034, -61.499, -78.87, 60.74, 67.962, -33.811]
  Call Extruder(8.09561)
  MoveL 3167 to (-39, 156.42, 59.84) mm, rotated rx 180 ry 0 rz -180 deg; joints [-126.042, -61.48, -78.921, 60.721, 67.973, -33.778]
  MoveL 3168 to (-39, 156.42, 59.84) mm, rotated rx 180 ry 0 rz -180 deg; joints [-126.042, -61.48, -78.921, 60.721, 67.973, -33.778]
  Call Extruder(8.25300)
  MoveL 3169 to (-39.1, 156.17, 59.84) mm, rotated rx 180 ry 0 rz -180 deg; joints [-126.05, -61.461, -78.972, 60.703, 67.985, -33.746]
  MoveL 3170 to (-39.1, 156.17, 59.84) mm, rotated rx 180 ry 0 rz -180 deg; joints [-126.05, -61.461, -78.972, 60.703, 67.985, -33.746]
  Call Extruder(8.43572)
  MoveL 3171 to (-39.23, 155.87, 59.84) mm, rotated rx -180 ry 0 rz -180 deg; joints [-126.06, -61.44, -79.031, 60.681, 67.997, -33.707]
  MoveL 3172 to (-39.23, 155.87, 59.84) mm, rotated rx -180 ry 0 rz -180 deg; joints [-126.06, -61.44, -79.031, 60.681, 67.997, -33.707]
  Call Extruder(8.61768)
  MoveL 3173 to (-39.35, 155.58, 59.84) mm, rotated rx 180 ry 0 rz -180 deg; joints [-126.07, -61.418, -79.09, 60.659, 68.01, -33.669]
  MoveL 3174 to (-39.35, 155.58, 59.84) mm, rotated rx 180 ry 0 rz -180 deg; joints [-126.07, -61.418, -79.09, 60.659, 68.01, -33.669]
  Call Extruder(8.76501)
  MoveL 3175 to (-39.44, 155.34, 59.84) mm, rotated rx 180 ry 0 rz 180 deg; joints [-126.079, -61.4, -79.138, 60.64, 68.02, -33.638]
  MoveL 3176 to (-39.44, 155.34, 59.84) mm, rotated rx 180 ry 0 rz 180 deg; joints [-126.079, -61.4, -79.138, 60.64, 68.02, -33.638]
  Call Extruder(8.87825)
  MoveL 3177 to (-39.5, 155.15, 59.84) mm, rotated rx 180 ry 0 rz -180 deg; joints [-126.087, -61.387, -79.174, 60.625, 68.027, -33.613]
  MoveL 3178 to (-39.5, 155.15, 59.84) mm, rotated rx 180 ry 0 rz -180 deg; joints [-126.087, -61.387, -79.174, 60.625, 68.027, -33.613]
  Call Extruder(8.99104)
  MoveL 3179 to (-39.56, 154.97, 59.84) mm, rotated rx -180 ry 0 rz -180 deg; joints [-126.095, -61.373, -79.21, 60.61, 68.033, -33.589]
  MoveL 3180 to (-39.56, 154.97, 59.84) mm, rotated rx -180 ry 0 rz -180 deg; joints [-126.095, -61.373, -79.21, 60.61, 68.033, -33.589]
  Call Extruder(9.10338)
  MoveL 3181 to (-39.62, 154.78, 59.84) mm, rotated rx 180 ry 0 rz -180 deg; joints [-126.103, -61.36, -79.246, 60.594, 68.04, -33.565]
  MoveL 3182 to (-39.62, 154.78, 59.84) mm, rotated rx 180 ry 0 rz -180 deg; joints [-126.103, -61.36, -79.246, 60.594, 68.04, -33.565]
  Call Extruder(9.21528)
  MoveL 3183 to (-39.68, 154.59, 59.84) mm, rotated rx 180 ry 0 rz -180 deg; joints [-126.111, -61.346, -79.283, 60.579, 68.047, -33.541]
  MoveL 3184 to (-39.68, 154.59, 59.84) mm, rotated rx 180 ry 0 rz -180 deg; joints [-126.111, -61.346, -79.283, 60.579, 68.047, -33.541]
  Call Extruder(9.33668)
  MoveL 3185 to (-39.75, 154.38, 59.84) mm, rotated rx -180 ry 0 rz 180 deg; joints [-126.12, -61.332, -79.322, 60.562, 68.054, -33.514]
  MoveL 3186 to (-39.75, 154.38, 59.84) mm, rotated rx -180 ry 0 rz 180 deg; joints [-126.12, -61.332, -79.322, 60.562, 68.054, -33.514]
  Call Extruder(9.46748)
  MoveL 3187 to (-39.82, 154.16, 59.84) mm, rotated rx 180 ry 0 rz -180 deg; joints [-126.131, -61.316, -79.364, 60.544, 68.061, -33.486]
  MoveL 3188 to (-39.82, 154.16, 59.84) mm, rotated rx 180 ry 0 rz -180 deg; joints [-126.131, -61.316, -79.364, 60.544, 68.061, -33.486]
  Call Extruder(9.59771)
  MoveL 3189 to (-39.88, 153.94, 59.84) mm, rotated rx 180 ry 0 rz 180 deg; joints [-126.141, -61.301, -79.406, 60.525, 68.069, -33.457]
  MoveL 3190 to (-39.88, 153.94, 59.84) mm, rotated rx 180 ry 0 rz 180 deg; joints [-126.141, -61.301, -79.406, 60.525, 68.069, -33.457]
  Call Extruder(9.72737)
  MoveL 3191 to (-39.95, 153.71, 59.84) mm, rotated rx 180 ry 0 rz -180 deg; joints [-126.151, -61.285, -79.449, 60.506, 68.076, -33.429]
  MoveL 3192 to (-39.95, 153.71, 59.84) mm, rotated rx 180 ry 0 rz -180 deg; joints [-126.151, -61.285, -79.449, 60.506, 68.076, -33.429]
  Call Extruder(9.85647)
  MoveL 3193 to (-40.02, 153.49, 59.84) mm, rotated rx 180 ry 0 rz 180 deg; joints [-126.161, -61.27, -79.491, 60.488, 68.084, -33.4]
  MoveL 3194 to (-40.02, 153.49, 59.84) mm, rotated rx 180 ry 0 rz 180 deg; joints [-126.161, -61.27, -79.491, 60.488, 68.084, -33.4]
  Call Extruder(9.97156)
  MoveL 3195 to (-40.06, 153.28, 59.84) mm, rotated rx -180 ry 0 rz 180 deg; joints [-126.173, -61.256, -79.528, 60.47, 68.089, -33.375]
  MoveL 3196 to (-40.06, 153.28, 59.84) mm, rotated rx -180 ry 0 rz 180 deg; joints [-126.173, -61.256, -79.528, 60.47, 68.089, -33.375]
  Call Extruder(10.08619)
  MoveL 3197 to (-40.11, 153.08, 59.84) mm, rotated rx -180 ry 0 rz 180 deg; joints [-126.184, -61.243, -79.564, 60.451, 68.094, -33.349]
  MoveL 3198 to (-40.11, 153.08, 59.84) mm, rotated rx -180 ry 0 rz 180 deg; joints [-126.184, -61.243, -79.564, 60.451, 68.094, -33.349]
  Call Extruder(10.20037)
  MoveL 3199 to (-40.15, 152.88, 59.84) mm, rotated rx 180 ry 0 rz 180 deg; joints [-126.195, -61.229, -79.601, 60.433, 68.1, -33.324]
  MoveL 3200 to (-40.15, 152.88, 59.84) mm, rotated rx 180 ry 0 rz 180 deg; joints [-126.195, -61.229, -79.601, 60.433, 68.1, -33.324]
  Call Extruder(10.31410)
  MoveL 3201 to (-40.2, 152.67, 59.84) mm, rotated rx -180 ry 0 rz 180 deg; joints [-126.206, -61.216, -79.638, 60.415, 68.105, -33.298]
  MoveL 3202 to (-40.2, 152.67, 59.84) mm, rotated rx -180 ry 0 rz 180 deg; joints [-126.206, -61.216, -79.638, 60.415, 68.105, -33.298]
  Call Extruder(10.43953)
  MoveL 3203 to (-40.24, 152.44, 59.84) mm, rotated rx -180 ry 0 rz 180 deg; joints [-126.219, -61.201, -79.678, 60.394, 68.11, -33.27]
  MoveL 3204 to (-40.24, 152.44, 59.84) mm, rotated rx -180 ry 0 rz 180 deg; joints [-126.219, -61.201, -79.678, 60.394, 68.11, -33.27]
  Call Extruder(10.57650)
  MoveL 3205 to (-40.29, 152.2, 59.84) mm, rotated rx 180 ry 0 rz 180 deg; joints [-126.233, -61.185, -79.722, 60.372, 68.116, -33.239]
  MoveL 3206 to (-40.29, 152.2, 59.84) mm, rotated rx 180 ry 0 rz 180 deg; joints [-126.233, -61.185, -79.722, 60.372, 68.116, -33.239]
  Call Extruder(10.71287)
  MoveL 3207 to (-40.34, 151.95, 59.84) mm, rotated rx 180 ry 0 rz 180 deg; joints [-126.248, -61.168, -79.766, 60.349, 68.122, -33.208]
  MoveL 3208 to (-40.34, 151.95, 59.84) mm, rotated rx 180 ry 0 rz 180 deg; joints [-126.248, -61.168, -79.766, 60.349, 68.122, -33.208]
  Call Extruder(10.84862)
  MoveL 3209 to (-40.39, 151.7, 59.84) mm, rotated rx 180 ry 0 rz -180 deg; joints [-126.262, -61.152, -79.81, 60.327, 68.128, -33.177]
  MoveL 3210 to (-40.39, 151.7, 59.84) mm, rotated rx 180 ry 0 rz -180 deg; joints [-126.262, -61.152, -79.81, 60.327, 68.128, -33.177]
  Call Extruder(10.98377)
  MoveL 3211 to (-40.44, 151.45, 59.84) mm, rotated rx 180 ry 0 rz 180 deg; joints [-126.276, -61.136, -79.854, 60.304, 68.134, -33.147]
  MoveL 3212 to (-40.44, 151.45, 59.84) mm, rotated rx 180 ry 0 rz 180 deg; joints [-126.276, -61.136, -79.854, 60.304, 68.134, -33.147]
  Call Extruder(11.11831)
  MoveL 3213 to (-40.49, 151.2, 59.84) mm, rotated rx -180 ry 0 rz 180 deg; joints [-126.291, -61.12, -79.898, 60.281, 68.14, -33.116]
  MoveL 3214 to (-40.49, 151.2, 59.84) mm, rotated rx -180 ry 0 rz 180 deg; joints [-126.291, -61.12, -79.898, 60.281, 68.14, -33.116]
  Call Extruder(11.25223)
  MoveL 3215 to (-40.54, 150.95, 59.84) mm, rotated rx 180 ry 0 rz -180 deg; joints [-126.305, -61.104, -79.942, 60.259, 68.146, -33.085]
  MoveL 3216 to (-40.54, 150.95, 59.84) mm, rotated rx 180 ry 0 rz -180 deg; joints [-126.305, -61.104, -79.942, 60.259, 68.146, -33.085]
  Call Extruder(11.40009)
  MoveL 3217 to (-40.59, 150.67, 59.84) mm, rotated rx 180 ry 0 rz 180 deg; joints [-126.322, -61.086, -79.99, 60.233, 68.152, -33.051]
  MoveL 3218 to (-40.59, 150.67, 59.84) mm, rotated rx 180 ry 0 rz 180 deg; joints [-126.322, -61.086, -79.99, 60.233, 68.152, -33.051]
  Call Extruder(11.56181)
  MoveL 3219 to (-40.64, 150.37, 59.84) mm, rotated rx 180 ry 0 rz 180 deg; joints [-126.341, -61.067, -80.043, 60.204, 68.158, -33.013]
  MoveL 3220 to (-40.64, 150.37, 59.84) mm, rotated rx 180 ry 0 rz 180 deg; joints [-126.341, -61.067, -80.043, 60.204, 68.158, -33.013]
  Call Extruder(11.72281)
  MoveL 3221 to (-40.69, 150.06, 59.84) mm, rotated rx 180 ry 0 rz -180 deg; joints [-126.36, -61.048, -80.095, 60.176, 68.165, -32.976]
  MoveL 3222 to (-40.69, 150.06, 59.84) mm, rotated rx 180 ry 0 rz -180 deg; joints [-126.36, -61.048, -80.095, 60.176, 68.165, -32.976]
  Call Extruder(11.88308)
  MoveL 3223 to (-40.74, 149.76, 59.84) mm, rotated rx 180 ry 0 rz 180 deg; joints [-126.379, -61.029, -80.148, 60.147, 68.171, -32.938]
  MoveL 3224 to (-40.74, 149.76, 59.84) mm, rotated rx 180 ry 0 rz 180 deg; joints [-126.379, -61.029, -80.148, 60.147, 68.171, -32.938]
  Call Extruder(12.04262)
  MoveL 3225 to (-40.78, 149.45, 59.84) mm, rotated rx 180 ry 0 rz 180 deg; joints [-126.398, -61.01, -80.2, 60.118, 68.177, -32.901]
  MoveL 3226 to (-40.78, 149.45, 59.84) mm, rotated rx 180 ry 0 rz 180 deg; joints [-126.398, -61.01, -80.2, 60.118, 68.177, -32.901]
  Call Extruder(12.20144)
  MoveL 3227 to (-40.83, 149.14, 59.84) mm, rotated rx -180 ry 0 rz 180 deg; joints [-126.417, -60.991, -80.252, 60.089, 68.183, -32.863]
  MoveL 3228 to (-40.83, 149.14, 59.84) mm, rotated rx -180 ry 0 rz 180 deg; joints [-126.417, -60.991, -80.252, 60.089, 68.183, -32.863]
  Call Extruder(12.38010)
  MoveL 3229 to (-40.88, 148.8, 59.84) mm, rotated rx -180 ry 0 rz 180 deg; joints [-126.439, -60.969, -80.311, 60.056, 68.19, -32.821]
  MoveL 3230 to (-40.88, 148.8, 59.84) mm, rotated rx -180 ry 0 rz 180 deg; joints [-126.439, -60.969, -80.311, 60.056, 68.19, -32.821]
  Call Extruder(12.57854)
  MoveL 3231 to (-40.92, 148.41, 59.84) mm, rotated rx -180 ry 0 rz 180 deg; joints [-126.465, -60.946, -80.375, 60.018, 68.196, -32.774]
  MoveL 3232 to (-40.92, 148.41, 59.84) mm, rotated rx -180 ry 0 rz 180 deg; joints [-126.465, -60.946, -80.375, 60.018, 68.196, -32.774]
  Call Extruder(12.77612)
  MoveL 3233 to (-40.97, 148.02, 59.84) mm, rotated rx 180 ry 0 rz -180 deg; joints [-126.491, -60.922, -80.44, 59.981, 68.202, -32.727]
  MoveL 3234 to (-40.97, 148.02, 59.84) mm, rotated rx 180 ry 0 rz -180 deg; joints [-126.491, -60.922, -80.44, 59.981, 68.202, -32.727]
  Call Extruder(12.97282)
  MoveL 3235 to (-41.02, 147.63, 59.84) mm, rotated rx -180 ry 0 rz -180 deg; joints [-126.517, -60.899, -80.504, 59.943, 68.209, -32.68]
  MoveL 3236 to (-41.02, 147.63, 59.84) mm, rotated rx -180 ry 0 rz -180 deg; joints [-126.517, -60.899, -80.504, 59.943, 68.209, -32.68]
  Call Extruder(13.16866)
  MoveL 3237 to (-41.06, 147.25, 59.84) mm, rotated rx 180 ry 0 rz 180 deg; joints [-126.543, -60.876, -80.568, 59.905, 68.215, -32.633]
  MoveL 3238 to (-41.06, 147.25, 59.84) mm, rotated rx 180 ry 0 rz 180 deg; joints [-126.543, -60.876, -80.568, 59.905, 68.215, -32.633]
  Call Extruder(13.46406)
  MoveL 3239 to (-41.11, 146.66, 59.84) mm, rotated rx 180 ry 0 rz -180 deg; joints [-126.585, -60.841, -80.663, 59.846, 68.223, -32.563]
  MoveL 3240 to (-41.11, 146.66, 59.84) mm, rotated rx 180 ry 0 rz -180 deg; joints [-126.585, -60.841, -80.663, 59.846, 68.223, -32.563]
  Call Extruder(13.75812)
  MoveL 3241 to (-41.15, 146.07, 59.84) mm, rotated rx 180 ry 0 rz 180 deg; joints [-126.628, -60.807, -80.758, 59.786, 68.231, -32.492]
  MoveL 3242 to (-41.15, 146.07, 59.84) mm, rotated rx 180 ry 0 rz 180 deg; joints [-126.628, -60.807, -80.758, 59.786, 68.231, -32.492]
  Call Extruder(14.05086)
  MoveL 3243 to (-41.2, 145.48, 59.84) mm, rotated rx 180 ry 0 rz 180 deg; joints [-126.67, -60.772, -80.853, 59.727, 68.238, -32.422]
  MoveL 3244 to (-41.2, 145.48, 59.84) mm, rotated rx 180 ry 0 rz 180 deg; joints [-126.67, -60.772, -80.853, 59.727, 68.238, -32.422]
  Call Extruder(14.62431)
  MoveL 3245 to (-41.25, 144.32, 59.84) mm, rotated rx 180 ry 0 rz 180 deg; joints [-126.759, -60.707, -81.035, 59.606, 68.249, -32.284]
  MoveL 3246 to (-41.25, 144.32, 59.84) mm, rotated rx 180 ry 0 rz 180 deg; joints [-126.759, -60.707, -81.035, 59.606, 68.249, -32.284]
  Call Extruder(15.33827)
  MoveL 3247 to (-41.29, 142.86, 59.84) mm, rotated rx 180 ry 0 rz -180 deg; joints [-126.873, -60.626, -81.259, 59.453, 68.261, -32.113]
  Call Extruder(57.40310)
  MoveL 3248 to (-41.29, 57.14, 59.84) mm, rotated rx 180 ry 0 rz 180 deg; joints [-135.148, -56.807, -92.846, 49.06, 69.012, -22.436]
  Call Extruder(57.83165)
  MoveL 3249 to (-41.27, 56.26, 59.84) mm, rotated rx 180 ry 0 rz -180 deg; joints [-135.25, -56.777, -92.948, 48.938, 69.021, -22.341]
  MoveL 3250 to (-41.27, 56.26, 59.84) mm, rotated rx 180 ry 0 rz -180 deg; joints [-135.25, -56.777, -92.948, 48.938, 69.021, -22.341]
  Call Extruder(58.11773)
  MoveL 3251 to (-41.25, 55.68, 59.84) mm, rotated rx 180 ry 0 rz 180 deg; joints [-135.318, -56.758, -93.015, 48.857, 69.025, -22.279]
  MoveL 3252 to (-41.25, 55.68, 59.84) mm, rotated rx 180 ry 0 rz 180 deg; joints [-135.318, -56.758, -93.015, 48.857, 69.025, -22.279]
  Call Extruder(58.69247)
  MoveL 3253 to (-41.2, 54.52, 59.84) mm, rotated rx 180 ry 0 rz 180 deg; joints [-135.457, -56.719, -93.148, 48.692, 69.035, -22.154]
  MoveL 3254 to (-41.2, 54.52, 59.84) mm, rotated rx 180 ry 0 rz 180 deg; joints [-135.457, -56.719, -93.148, 48.692, 69.035, -22.154]
  Call Extruder(58.98587)
  MoveL 3255 to (-41.16, 53.93, 59.84) mm, rotated rx -180 ry 0 rz 180 deg; joints [-135.53, -56.7, -93.212, 48.607, 69.038, -22.092]
  MoveL 3256 to (-41.16, 53.93, 59.84) mm, rotated rx -180 ry 0 rz 180 deg; joints [-135.53, -56.7, -93.212, 48.607, 69.038, -22.092]
  Call Extruder(59.28060)
  MoveL 3257 to (-41.11, 53.34, 59.84) mm, rotated rx 180 ry 0 rz -180 deg; joints [-135.603, -56.681, -93.276, 48.521, 69.04, -22.029]
  MoveL 3258 to (-41.11, 53.34, 59.84) mm, rotated rx 180 ry 0 rz -180 deg; joints [-135.603, -56.681, -93.276, 48.521, 69.04, -22.029]
  Call Extruder(59.57666)
  MoveL 3259 to (-41.06, 52.75, 59.84) mm, rotated rx 180 ry 0 rz 180 deg; joints [-135.676, -56.663, -93.34, 48.435, 69.043, -21.967]
  MoveL 3260 to (-41.06, 52.75, 59.84) mm, rotated rx 180 ry 0 rz 180 deg; joints [-135.676, -56.663, -93.34, 48.435, 69.043, -21.967]
  Call Extruder(59.77294)
  MoveL 3261 to (-41.02, 52.37, 59.84) mm, rotated rx 180 ry 0 rz 180 deg; joints [-135.726, -56.651, -93.38, 48.377, 69.043, -21.926]
  MoveL 3262 to (-41.02, 52.37, 59.84) mm, rotated rx 180 ry 0 rz 180 deg; joints [-135.726, -56.651, -93.38, 48.377, 69.043, -21.926]
  Call Extruder(59.97008)
  MoveL 3263 to (-40.97, 51.98, 59.84) mm, rotated rx 180 ry 0 rz 180 deg; joints [-135.776, -56.64, -93.421, 48.319, 69.043, -21.885]
  MoveL 3264 to (-40.97, 51.98, 59.84) mm, rotated rx 180 ry 0 rz 180 deg; joints [-135.776, -56.64, -93.421, 48.319, 69.043, -21.885]
  Call Extruder(60.16808)
  MoveL 3265 to (-40.92, 51.59, 59.84) mm, rotated rx 180 ry 0 rz -180 deg; joints [-135.827, -56.628, -93.461, 48.261, 69.044, -21.845]
  MoveL 3266 to (-40.92, 51.59, 59.84) mm, rotated rx 180 ry 0 rz -180 deg; joints [-135.827, -56.628, -93.461, 48.261, 69.044, -21.845]
  Call Extruder(60.36696)
  MoveL 3267 to (-40.88, 51.2, 59.84) mm, rotated rx -180 ry 0 rz 180 deg; joints [-135.877, -56.616, -93.501, 48.203, 69.044, -21.804]
  MoveL 3268 to (-40.88, 51.2, 59.84) mm, rotated rx -180 ry 0 rz 180 deg; joints [-135.877, -56.616, -93.501, 48.203, 69.044, -21.804]
  Call Extruder(60.54604)
  MoveL 3269 to (-40.83, 50.86, 59.84) mm, rotated rx 180 ry 0 rz 180 deg; joints [-135.922, -56.606, -93.536, 48.151, 69.044, -21.768]
  MoveL 3270 to (-40.83, 50.86, 59.84) mm, rotated rx 180 ry 0 rz 180 deg; joints [-135.922, -56.606, -93.536, 48.151, 69.044, -21.768]
  Call Extruder(60.70522)
  MoveL 3271 to (-40.78, 50.55, 59.84) mm, rotated rx 180 ry 0 rz 180 deg; joints [-135.964, -56.598, -93.565, 48.104, 69.043, -21.737]
  MoveL 3272 to (-40.78, 50.55, 59.84) mm, rotated rx 180 ry 0 rz 180 deg; joints [-135.964, -56.598, -93.565, 48.104, 69.043, -21.737]
  Call Extruder(60.86512)
  MoveL 3273 to (-40.73, 50.24, 59.84) mm, rotated rx 180 ry 0 rz 180 deg; joints [-136.005, -56.589, -93.595, 48.057, 69.042, -21.705]
  MoveL 3274 to (-40.73, 50.24, 59.84) mm, rotated rx 180 ry 0 rz 180 deg; joints [-136.005, -56.589, -93.595, 48.057, 69.042, -21.705]
  Call Extruder(61.02576)
  MoveL 3275 to (-40.69, 49.94, 59.84) mm, rotated rx -180 ry 0 rz -180 deg; joints [-136.046, -56.581, -93.625, 48.01, 69.041, -21.673]
  MoveL 3276 to (-40.69, 49.94, 59.84) mm, rotated rx -180 ry 0 rz -180 deg; joints [-136.046, -56.581, -93.625, 48.01, 69.041, -21.673]
  Call Extruder(61.18712)
  MoveL 3277 to (-40.64, 49.63, 59.84) mm, rotated rx 180 ry 0 rz 180 deg; joints [-136.087, -56.572, -93.655, 47.963, 69.04, -21.642]
  MoveL 3278 to (-40.64, 49.63, 59.84) mm, rotated rx 180 ry 0 rz 180 deg; joints [-136.087, -56.572, -93.655, 47.963, 69.04, -21.642]
  Call Extruder(61.34921)
  MoveL 3279 to (-40.59, 49.33, 59.84) mm, rotated rx 180 ry 0 rz 180 deg; joints [-136.128, -56.563, -93.685, 47.916, 69.039, -21.61]
  MoveL 3280 to (-40.59, 49.33, 59.84) mm, rotated rx 180 ry 0 rz 180 deg; joints [-136.128, -56.563, -93.685, 47.916, 69.039, -21.61]
  Call Extruder(61.49741)
  MoveL 3281 to (-40.54, 49.05, 59.84) mm, rotated rx 180 ry 0 rz 180 deg; joints [-136.166, -56.556, -93.711, 47.872, 69.037, -21.582]
  MoveL 3282 to (-40.54, 49.05, 59.84) mm, rotated rx 180 ry 0 rz 180 deg; joints [-136.166, -56.556, -93.711, 47.872, 69.037, -21.582]
  Call Extruder(61.63164)
  MoveL 3283 to (-40.49, 48.8, 59.84) mm, rotated rx -180 ry 0 rz -180 deg; joints [-136.201, -56.549, -93.734, 47.833, 69.035, -21.556]
  MoveL 3284 to (-40.49, 48.8, 59.84) mm, rotated rx -180 ry 0 rz -180 deg; joints [-136.201, -56.549, -93.734, 47.833, 69.035, -21.556]
  Call Extruder(61.76648)
  MoveL 3285 to (-40.44, 48.55, 59.84) mm, rotated rx 180 ry 0 rz -180 deg; joints [-136.236, -56.543, -93.757, 47.794, 69.034, -21.531]
  MoveL 3286 to (-40.44, 48.55, 59.84) mm, rotated rx 180 ry 0 rz -180 deg; joints [-136.236, -56.543, -93.757, 47.794, 69.034, -21.531]
  Call Extruder(61.90193)
  MoveL 3287 to (-40.39, 48.3, 59.84) mm, rotated rx -180 ry 0 rz 180 deg; joints [-136.271, -56.536, -93.78, 47.754, 69.032, -21.505]
  MoveL 3288 to (-40.39, 48.3, 59.84) mm, rotated rx -180 ry 0 rz 180 deg; joints [-136.271, -56.536, -93.78, 47.754, 69.032, -21.505]
  Call Extruder(62.03799)
  MoveL 3289 to (-40.34, 48.05, 59.84) mm, rotated rx -180 ry 0 rz 180 deg; joints [-136.306, -56.529, -93.803, 47.715, 69.03, -21.48]
  MoveL 3290 to (-40.34, 48.05, 59.84) mm, rotated rx -180 ry 0 rz 180 deg; joints [-136.306, -56.529, -93.803, 47.715, 69.03, -21.48]
  Call Extruder(62.17466)
  MoveL 3291 to (-40.29, 47.8, 59.84) mm, rotated rx -180 ry 0 rz -180 deg; joints [-136.341, -56.523, -93.826, 47.675, 69.028, -21.455]
  MoveL 3292 to (-40.29, 47.8, 59.84) mm, rotated rx -180 ry 0 rz -180 deg; joints [-136.341, -56.523, -93.826, 47.675, 69.028, -21.455]
  Call Extruder(62.31194)
  MoveL 3293 to (-40.24, 47.55, 59.84) mm, rotated rx -180 ry 0 rz 180 deg; joints [-136.376, -56.516, -93.849, 47.636, 69.027, -21.429]
  MoveL 3294 to (-40.24, 47.55, 59.84) mm, rotated rx -180 ry 0 rz 180 deg; joints [-136.376, -56.516, -93.849, 47.636, 69.027, -21.429]
  Call Extruder(62.43761)
  MoveL 3295 to (-40.2, 47.33, 59.84) mm, rotated rx 180 ry 0 rz 180 deg; joints [-136.408, -56.51, -93.87, 47.6, 69.025, -21.406]
  MoveL 3296 to (-40.2, 47.33, 59.84) mm, rotated rx 180 ry 0 rz 180 deg; joints [-136.408, -56.51, -93.87, 47.6, 69.025, -21.406]
  Call Extruder(62.55157)
  MoveL 3297 to (-40.15, 47.12, 59.84) mm, rotated rx 180 ry 0 rz 180 deg; joints [-136.437, -56.505, -93.888, 47.567, 69.023, -21.385]
  MoveL 3298 to (-40.15, 47.12, 59.84) mm, rotated rx 180 ry 0 rz 180 deg; joints [-136.437, -56.505, -93.888, 47.567, 69.023, -21.385]
  Call Extruder(62.66597)
  MoveL 3299 to (-40.11, 46.92, 59.84) mm, rotated rx -180 ry 0 rz 180 deg; joints [-136.466, -56.5, -93.906, 47.534, 69.021, -21.365]
  MoveL 3300 to (-40.11, 46.92, 59.84) mm, rotated rx -180 ry 0 rz 180 deg; joints [-136.466, -56.5, -93.906, 47.534, 69.021, -21.365]
  Call Extruder(62.78083)
  MoveL 3301 to (-40.06, 46.72, 59.84) mm, rotated rx 180 ry 0 rz -180 deg; joints [-136.495, -56.495, -93.924, 47.502, 69.019, -21.344]
  MoveL 3302 to (-40.06, 46.72, 59.84) mm, rotated rx 180 ry 0 rz -180 deg; joints [-136.495, -56.495, -93.924, 47.502, 69.019, -21.344]
  Call Extruder(62.89615)
  MoveL 3303 to (-40.02, 46.51, 59.84) mm, rotated rx 180 ry 0 rz 180 deg; joints [-136.525, -56.49, -93.942, 47.469, 69.017, -21.323]
  MoveL 3304 to (-40.02, 46.51, 59.84) mm, rotated rx 180 ry 0 rz 180 deg; joints [-136.525, -56.49, -93.942, 47.469, 69.017, -21.323]
  Call Extruder(63.02553)
  MoveL 3305 to (-39.95, 46.29, 59.84) mm, rotated rx 180 ry 0 rz -180 deg; joints [-136.559, -56.485, -93.96, 47.431, 69.013, -21.301]
  MoveL 3306 to (-39.95, 46.29, 59.84) mm, rotated rx 180 ry 0 rz -180 deg; joints [-136.559, -56.485, -93.96, 47.431, 69.013, -21.301]
  Call Extruder(63.15547)
  MoveL 3307 to (-39.88, 46.06, 59.84) mm, rotated rx -180 ry 0 rz -180 deg; joints [-136.593, -56.48, -93.978, 47.394, 69.01, -21.279]
  MoveL 3308 to (-39.88, 46.06, 59.84) mm, rotated rx -180 ry 0 rz -180 deg; joints [-136.593, -56.48, -93.978, 47.394, 69.01, -21.279]
  Call Extruder(63.28598)
  MoveL 3309 to (-39.81, 45.84, 59.84) mm, rotated rx 180 ry 0 rz 180 deg; joints [-136.627, -56.475, -93.995, 47.356, 69.006, -21.257]
  MoveL 3310 to (-39.81, 45.84, 59.84) mm, rotated rx 180 ry 0 rz 180 deg; joints [-136.627, -56.475, -93.995, 47.356, 69.006, -21.257]
  Call Extruder(63.41706)
  MoveL 3311 to (-39.75, 45.62, 59.84) mm, rotated rx 180 ry 0 rz 180 deg; joints [-136.661, -56.47, -94.013, 47.318, 69.002, -21.235]
  MoveL 3312 to (-39.75, 45.62, 59.84) mm, rotated rx 180 ry 0 rz 180 deg; joints [-136.661, -56.47, -94.013, 47.318, 69.002, -21.235]
  Call Extruder(63.53870)
  MoveL 3313 to (-39.68, 45.41, 59.84) mm, rotated rx 180 ry 0 rz 180 deg; joints [-136.693, -56.465, -94.029, 47.283, 68.998, -21.215]
  MoveL 3314 to (-39.68, 45.41, 59.84) mm, rotated rx 180 ry 0 rz 180 deg; joints [-136.693, -56.465, -94.029, 47.283, 68.998, -21.215]
  Call Extruder(63.65083)
  MoveL 3315 to (-39.62, 45.22, 59.84) mm, rotated rx -180 ry 0 rz 180 deg; joints [-136.722, -56.461, -94.043, 47.251, 68.994, -21.196]
  MoveL 3316 to (-39.62, 45.22, 59.84) mm, rotated rx -180 ry 0 rz 180 deg; joints [-136.722, -56.461, -94.043, 47.251, 68.994, -21.196]
  Call Extruder(63.76340)
  MoveL 3317 to (-39.56, 45.03, 59.84) mm, rotated rx 180 ry 0 rz -180 deg; joints [-136.751, -56.457, -94.057, 47.219, 68.991, -21.178]
  MoveL 3318 to (-39.56, 45.03, 59.84) mm, rotated rx 180 ry 0 rz -180 deg; joints [-136.751, -56.457, -94.057, 47.219, 68.991, -21.178]
  Call Extruder(63.87641)
  MoveL 3319 to (-39.5, 44.85, 59.84) mm, rotated rx 180 ry 0 rz -180 deg; joints [-136.781, -56.453, -94.071, 47.187, 68.987, -21.159]
  MoveL 3320 to (-39.5, 44.85, 59.84) mm, rotated rx 180 ry 0 rz -180 deg; joints [-136.781, -56.453, -94.071, 47.187, 68.987, -21.159]
  Call Extruder(63.98987)
  MoveL 3321 to (-39.44, 44.66, 59.84) mm, rotated rx 180 ry 0 rz -180 deg; joints [-136.81, -56.449, -94.085, 47.155, 68.983, -21.141]
  MoveL 3322 to (-39.44, 44.66, 59.84) mm, rotated rx 180 ry 0 rz -180 deg; joints [-136.81, -56.449, -94.085, 47.155, 68.983, -21.141]
  Call Extruder(64.13751)
  MoveL 3323 to (-39.35, 44.42, 59.84) mm, rotated rx 180 ry 0 rz 180 deg; joints [-136.849, -56.444, -94.102, 47.113, 68.977, -21.118]
  MoveL 3324 to (-39.35, 44.42, 59.84) mm, rotated rx 180 ry 0 rz 180 deg; joints [-136.849, -56.444, -94.102, 47.113, 68.977, -21.118]
  Call Extruder(64.31985)
